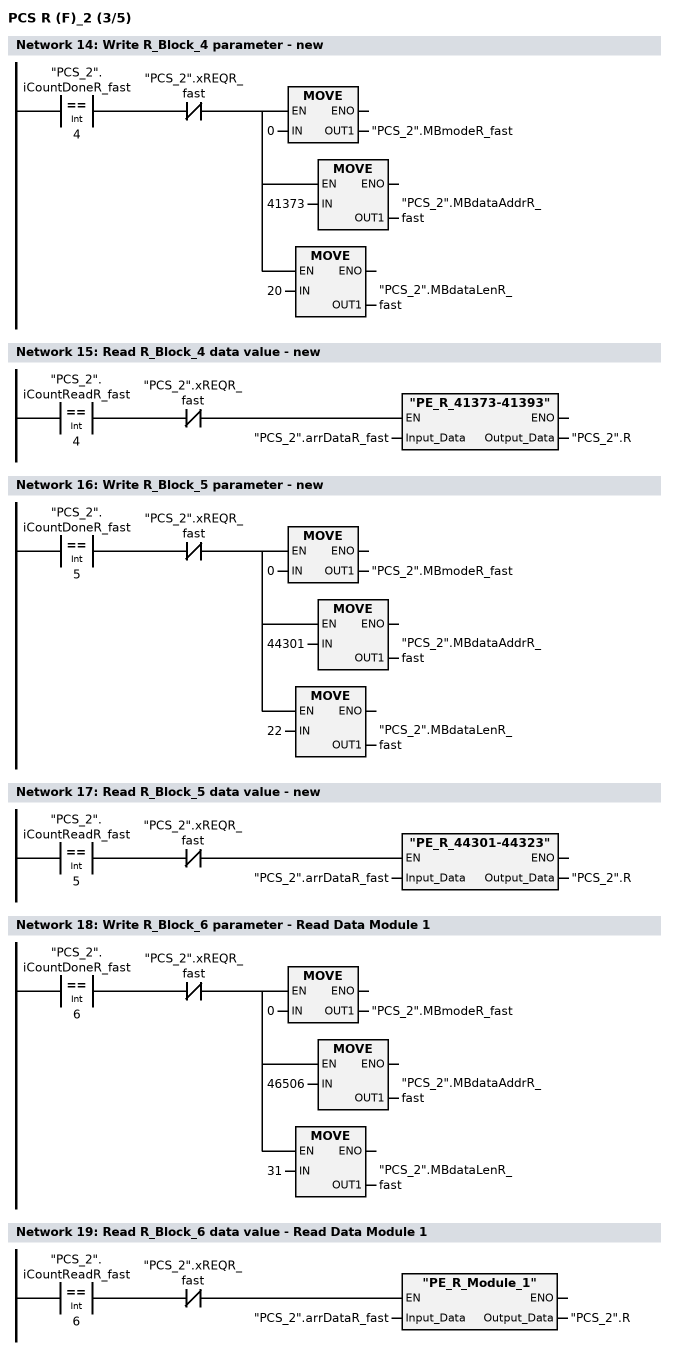
   RUNG wire#powerrail
      { S7_Templates := "SrcType := Int" } EQ_Contact(in1 := "PCS_2".iCountDoneR_fast, in2 := 4)
      I_Contact( "PCS_2".xREQR_fast )
      wire#w1
      Move(in := 0, out1 => "PCS_2".MBmodeR_fast)
   END_RUNG
   RUNG wire#w1
      Move(in := 41373, out1 => "PCS_2".MBdataAddrR_fast)
   END_RUNG
   RUNG wire#w1
      Move(in := 20, out1 => "PCS_2".MBdataLenR_fast)
   END_RUNG
   // the same network as SCL:
   IF ("PCS_2".iCountDoneR_fast = 4) AND NOT "PCS_2".xREQR_fast THEN
       "PCS_2".MBmodeR_fast := 0;
       "PCS_2".MBdataAddrR_fast := 41373;
       "PCS_2".MBdataLenR_fast := 20;
   END_IF;
END_REGION

REGION Network 15: Read R_Block_4 data value - new
   RUNG wire#powerrail
      { S7_Templates := "SrcType := Int" } EQ_Contact(in1 := "PCS_2".iCountReadR_fast, in2 := 4)
      I_Contact( "PCS_2".xREQR_fast )
      "PE_R_41373-41393"(Input_Data := "PCS_2".arrDataR_fast, Output_Data => "PCS_2".R)
   END_RUNG
   // the same network as SCL:
   IF ("PCS_2".iCountReadR_fast = 4) AND NOT "PCS_2".xREQR_fast THEN
       "PE_R_41373-41393"(Input_Data := "PCS_2".arrDataR_fast, Output_Data => "PCS_2".R);
   END_IF;
END_REGION

REGION Network 16: Write R_Block_5 parameter - new
   RUNG wire#powerrail
      { S7_Templates := "SrcType := Int" } EQ_Contact(in1 := "PCS_2".iCountDoneR_fast, in2 := 5)
      I_Contact( "PCS_2".xREQR_fast )
      wire#w1
      Move(in := 0, out1 => "PCS_2".MBmodeR_fast)
   END_RUNG
   RUNG wire#w1
      Move(in := 44301, out1 => "PCS_2".MBdataAddrR_fast)
   END_RUNG
   RUNG wire#w1
      Move(in := 22, out1 => "PCS_2".MBdataLenR_fast)
   END_RUNG
   // the same network as SCL:
   IF ("PCS_2".iCountDoneR_fast = 5) AND NOT "PCS_2".xREQR_fast THEN
       "PCS_2".MBmodeR_fast := 0;
       "PCS_2".MBdataAddrR_fast := 44301;
       "PCS_2".MBdataLenR_fast := 22;
   END_IF;
END_REGION

REGION Network 17: Read R_Block_5 data value - new
   RUNG wire#powerrail
      { S7_Templates := "SrcType := Int" } EQ_Contact(in1 := "PCS_2".iCountReadR_fast, in2 := 5)
      I_Contact( "PCS_2".xREQR_fast )
      "PE_R_44301-44323"(Input_Data := "PCS_2".arrDataR_fast, Output_Data => "PCS_2".R)
   END_RUNG
   // the same network as SCL:
   IF ("PCS_2".iCountReadR_fast = 5) AND NOT "PCS_2".xREQR_fast THEN
       "PE_R_44301-44323"(Input_Data := "PCS_2".arrDataR_fast, Output_Data => "PCS_2".R);
   END_IF;
END_REGION

REGION Network 18: Write R_Block_6 parameter - Read Data Module 1
   RUNG wire#powerrail
      { S7_Templates := "SrcType := Int" } EQ_Contact(in1 := "PCS_2".iCountDoneR_fast, in2 := 6)
      I_Contact( "PCS_2".xREQR_fast )
      wire#w1
      Move(in := 0, out1 => "PCS_2".MBmodeR_fast)
   END_RUNG
   RUNG wire#w1
      Move(in := 46506, out1 => "PCS_2".MBdataAddrR_fast)
   END_RUNG
   RUNG wire#w1
      Move(in := 31, out1 => "PCS_2".MBdataLenR_fast)
   END_RUNG
   // the same network as SCL:
   IF ("PCS_2".iCountDoneR_fast = 6) AND NOT "PCS_2".xREQR_fast THEN
       "PCS_2".MBmodeR_fast := 0;
       "PCS_2".MBdataAddrR_fast := 46506;
       "PCS_2".MBdataLenR_fast := 31;
   END_IF;
END_REGION

REGION Network 19: Read R_Block_6 data value - Read Data Module 1
   RUNG wire#powerrail
      { S7_Templates := "SrcType := Int" } EQ_Contact(in1 := "PCS_2".iCountReadR_fast, in2 := 6)
      I_Contact( "PCS_2".xREQR_fast )
      "PE_R_Module_1"(Input_Data := "PCS_2".arrDataR_fast, Output_Data => "PCS_2".R)
   END_RUNG
   // the same network as SCL:
   IF ("PCS_2".iCountReadR_fast = 6) AND NOT "PCS_2".xREQR_fast THEN
       "PE_R_Module_1"(Input_Data := "PCS_2".arrDataR_fast, Output_Data => "PCS_2".R);
   END_IF;
END_REGION

REGION Network 20: Write R_Block_7 parameter - Read Data Module 2
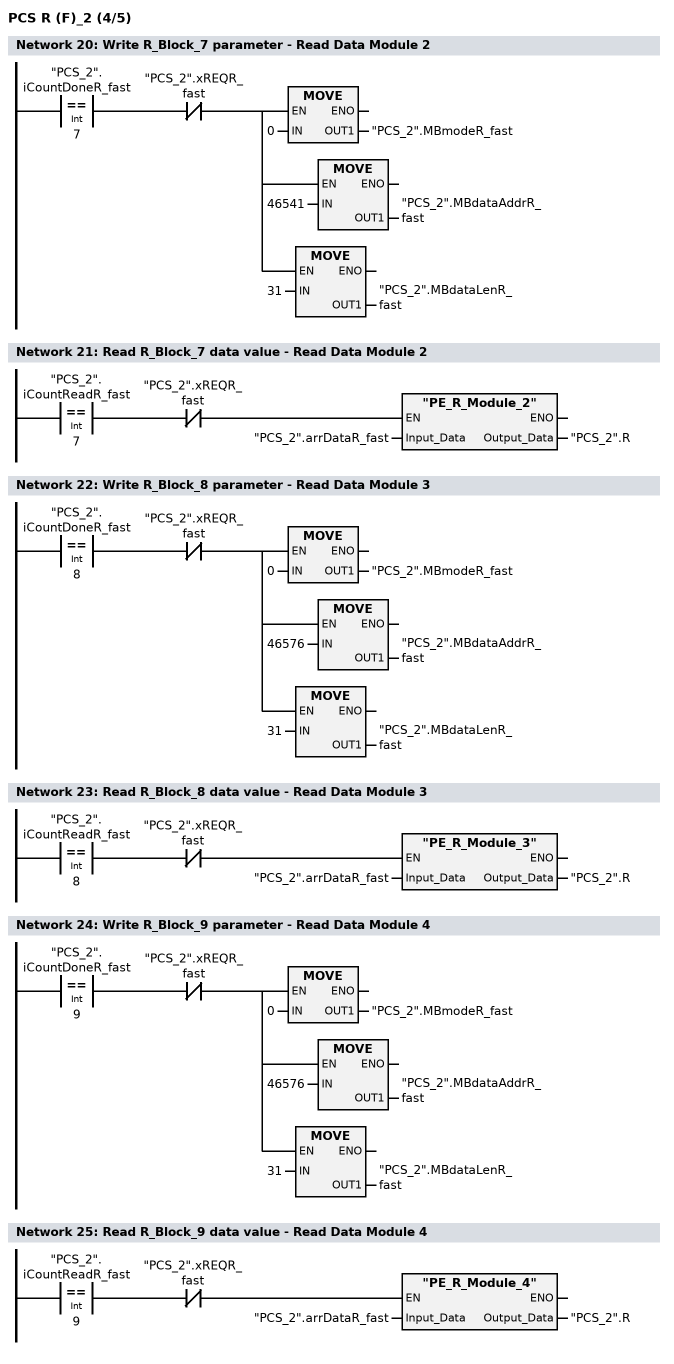
   RUNG wire#powerrail
      { S7_Templates := "SrcType := Int" } EQ_Contact(in1 := "PCS_2".iCountDoneR_fast, in2 := 7)
      I_Contact( "PCS_2".xREQR_fast )
      wire#w1
      Move(in := 0, out1 => "PCS_2".MBmodeR_fast)
   END_RUNG
   RUNG wire#w1
      Move(in := 46541, out1 => "PCS_2".MBdataAddrR_fast)
   END_RUNG
   RUNG wire#w1
      Move(in := 31, out1 => "PCS_2".MBdataLenR_fast)
   END_RUNG
   // the same network as SCL:
   IF ("PCS_2".iCountDoneR_fast = 7) AND NOT "PCS_2".xREQR_fast THEN
       "PCS_2".MBmodeR_fast := 0;
       "PCS_2".MBdataAddrR_fast := 46541;
       "PCS_2".MBdataLenR_fast := 31;
   END_IF;
END_REGION

REGION Network 21: Read R_Block_7 data value - Read Data Module 2
   RUNG wire#powerrail
      { S7_Templates := "SrcType := Int" } EQ_Contact(in1 := "PCS_2".iCountReadR_fast, in2 := 7)
      I_Contact( "PCS_2".xREQR_fast )
      "PE_R_Module_2"(Input_Data := "PCS_2".arrDataR_fast, Output_Data => "PCS_2".R)
   END_RUNG
   // the same network as SCL:
   IF ("PCS_2".iCountReadR_fast = 7) AND NOT "PCS_2".xREQR_fast THEN
       "PE_R_Module_2"(Input_Data := "PCS_2".arrDataR_fast, Output_Data => "PCS_2".R);
   END_IF;
END_REGION

REGION Network 22: Write R_Block_8 parameter - Read Data Module 3
   RUNG wire#powerrail
      { S7_Templates := "SrcType := Int" } EQ_Contact(in1 := "PCS_2".iCountDoneR_fast, in2 := 8)
      I_Contact( "PCS_2".xREQR_fast )
      wire#w1
      Move(in := 0, out1 => "PCS_2".MBmodeR_fast)
   END_RUNG
   RUNG wire#w1
      Move(in := 46576, out1 => "PCS_2".MBdataAddrR_fast)
   END_RUNG
   RUNG wire#w1
      Move(in := 31, out1 => "PCS_2".MBdataLenR_fast)
   END_RUNG
   // the same network as SCL:
   IF ("PCS_2".iCountDoneR_fast = 8) AND NOT "PCS_2".xREQR_fast THEN
       "PCS_2".MBmodeR_fast := 0;
       "PCS_2".MBdataAddrR_fast := 46576;
       "PCS_2".MBdataLenR_fast := 31;
   END_IF;
END_REGION

REGION Network 23: Read R_Block_8 data value - Read Data Module 3
   RUNG wire#powerrail
      { S7_Templates := "SrcType := Int" } EQ_Contact(in1 := "PCS_2".iCountReadR_fast, in2 := 8)
      I_Contact( "PCS_2".xREQR_fast )
      "PE_R_Module_3"(Input_Data := "PCS_2".arrDataR_fast, Output_Data => "PCS_2".R)
   END_RUNG
   // the same network as SCL:
   IF ("PCS_2".iCountReadR_fast = 8) AND NOT "PCS_2".xREQR_fast THEN
       "PE_R_Module_3"(Input_Data := "PCS_2".arrDataR_fast, Output_Data => "PCS_2".R);
   END_IF;
END_REGION

REGION Network 24: Write R_Block_9 parameter - Read Data Module 4
   RUNG wire#powerrail
      { S7_Templates := "SrcType := Int" } EQ_Contact(in1 := "PCS_2".iCountDoneR_fast, in2 := 9)
      I_Contact( "PCS_2".xREQR_fast )
      wire#w1
      Move(in := 0, out1 => "PCS_2".MBmodeR_fast)
   END_RUNG
   RUNG wire#w1
      Move(in := 46576, out1 => "PCS_2".MBdataAddrR_fast)
   END_RUNG
   RUNG wire#w1
      Move(in := 31, out1 => "PCS_2".MBdataLenR_fast)
   END_RUNG
   // the same network as SCL:
   IF ("PCS_2".iCountDoneR_fast = 9) AND NOT "PCS_2".xREQR_fast THEN
       "PCS_2".MBmodeR_fast := 0;
       "PCS_2".MBdataAddrR_fast := 46576;
       "PCS_2".MBdataLenR_fast := 31;
   END_IF;
END_REGION

REGION Network 25: Read R_Block_9 data value - Read Data Module 4
   RUNG wire#powerrail
      { S7_Templates := "SrcType := Int" } EQ_Contact(in1 := "PCS_2".iCountReadR_fast, in2 := 9)
      I_Contact( "PCS_2".xREQR_fast )
      "PE_R_Module_4"(Input_Data := "PCS_2".arrDataR_fast, Output_Data => "PCS_2".R)
   END_RUNG
   // the same network as SCL:
   IF ("PCS_2".iCountReadR_fast = 9) AND NOT "PCS_2".xREQR_fast THEN
       "PE_R_Module_4"(Input_Data := "PCS_2".arrDataR_fast, Output_Data => "PCS_2".R);
   END_IF;
END_REGION

REGION Network 26: Write R_Block_10 parameter - Read Humidity module 1-2-3-4
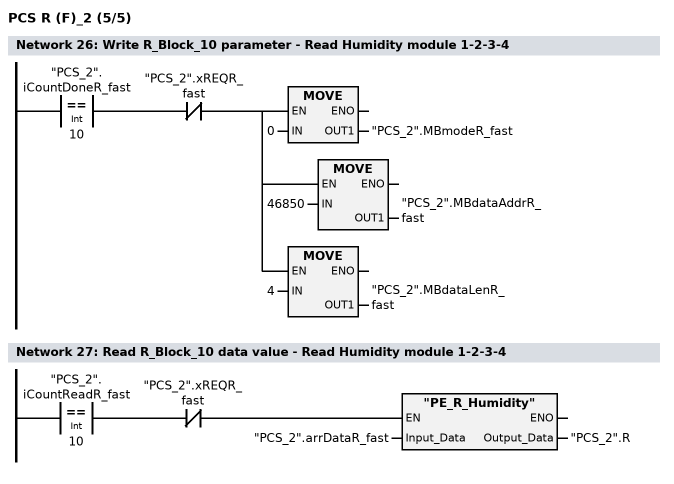
   RUNG wire#powerrail
      { S7_Templates := "SrcType := Int" } EQ_Contact(in1 := "PCS_2".iCountDoneR_fast, in2 := 10)
      I_Contact( "PCS_2".xREQR_fast )
      wire#w1
      Move(in := 0, out1 => "PCS_2".MBmodeR_fast)
   END_RUNG
   RUNG wire#w1
      Move(in := 46850, out1 => "PCS_2".MBdataAddrR_fast)
   END_RUNG
   RUNG wire#w1
      Move(in := 4, out1 => "PCS_2".MBdataLenR_fast)
   END_RUNG
   // the same network as SCL:
   IF ("PCS_2".iCountDoneR_fast = 10) AND NOT "PCS_2".xREQR_fast THEN
       "PCS_2".MBmodeR_fast := 0;
       "PCS_2".MBdataAddrR_fast := 46850;
       "PCS_2".MBdataLenR_fast := 4;
   END_IF;
END_REGION

REGION Network 27: Read R_Block_10 data value - Read Humidity module 1-2-3-4
   RUNG wire#powerrail
      { S7_Templates := "SrcType := Int" } EQ_Contact(in1 := "PCS_2".iCountReadR_fast, in2 := 10)
      I_Contact( "PCS_2".xREQR_fast )
      "PE_R_Humidity"(Input_Data := "PCS_2".arrDataR_fast, Output_Data => "PCS_2".R)
   END_RUNG
   // the same network as SCL:
   IF ("PCS_2".iCountReadR_fast = 10) AND NOT "PCS_2".xREQR_fast THEN
       "PE_R_Humidity"(Input_Data := "PCS_2".arrDataR_fast, Output_Data => "PCS_2".R);
   END_IF;
END_REGION
END_FUNCTION

FUNCTION "PCS R (S)_2" : Void   // FC49, LAD
TITLE = ModBus TCP for PCS Power Electronics
{ S7_Optimized_Access := 'TRUE' }
VERSION : 0.1
// stored: AutoNumber true, IsIECCheckEnabled false, SetENOAutomatically false, UDAEnableTagReadback false
   VAR_TEMP
      rVac : Real;
   END_VAR
   VAR_TEMP   // added for the SCL form of the ladder/FBD networks
      _w1 : Bool;
   END_VAR
BEGIN

REGION Network 1: Function Modbus Client
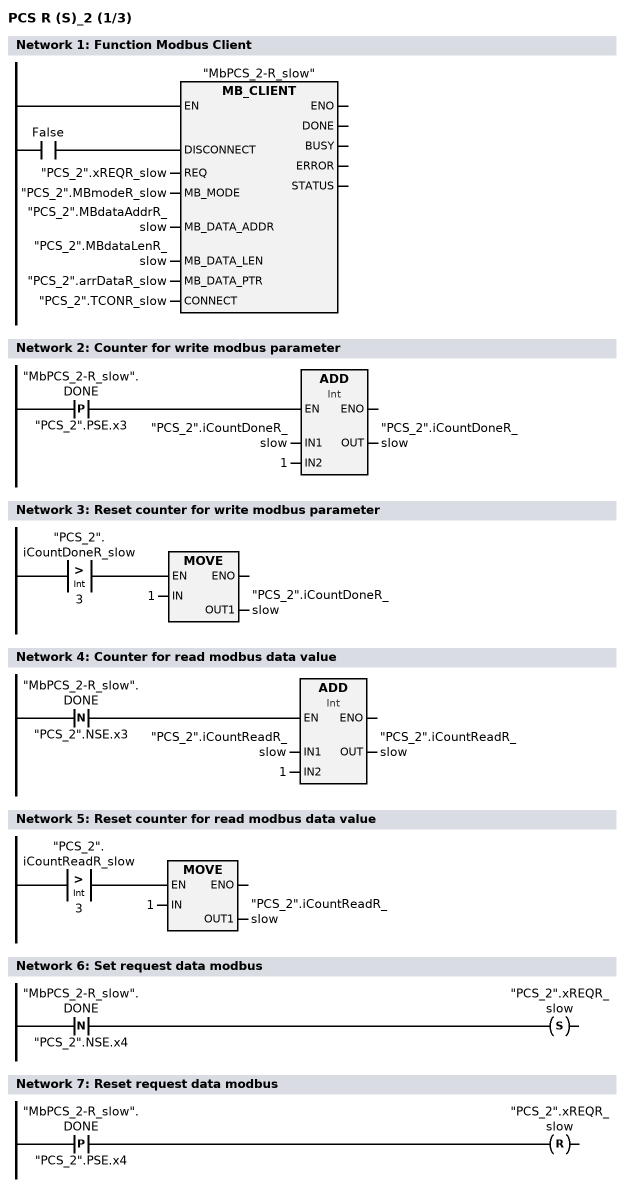
   RUNG wire#powerrail
      "MbPCS_2-R_slow".MB_CLIENT(DISCONNECT := wire#w1, REQ := "PCS_2".xREQR_slow, MB_MODE := "PCS_2".MBmodeR_slow, MB_DATA_ADDR := "PCS_2".MBdataAddrR_slow, MB_DATA_LEN := "PCS_2".MBdataLenR_slow, MB_DATA_PTR := "PCS_2".arrDataR_slow, CONNECT := "PCS_2".TCONR_slow, DONE =>, BUSY =>, ERROR =>, STATUS =>)
   END_RUNG
   RUNG wire#powerrail
      Contact( False )
   END_RUNG wire#w1
   // the same network as SCL:
   "MbPCS_2-R_slow"(DISCONNECT := False,   // MB_CLIENT
                    REQ := "PCS_2".xREQR_slow,
                    MB_MODE := "PCS_2".MBmodeR_slow,
                    MB_DATA_ADDR := "PCS_2".MBdataAddrR_slow,
                    MB_DATA_LEN := "PCS_2".MBdataLenR_slow,
                    MB_DATA_PTR := "PCS_2".arrDataR_slow,
                    CONNECT := "PCS_2".TCONR_slow);
END_REGION

REGION Network 2: Counter for write modbus parameter
   RUNG wire#powerrail
      P_Contact(operand := "MbPCS_2-R_slow".DONE, bit := "PCS_2".PSE.x3)
      { S7_Templates := "SrcType := Int" } Add(in1 := "PCS_2".iCountDoneR_slow, in2 := 1, out => "PCS_2".iCountDoneR_slow)
   END_RUNG
   // the same network as SCL:
   #_w1 := "MbPCS_2-R_slow".DONE AND NOT "PCS_2".PSE.x3;   // rising edge of "MbPCS_2-R_slow".DONE
   "PCS_2".PSE.x3 := "MbPCS_2-R_slow".DONE;
   IF #_w1 THEN "PCS_2".iCountDoneR_slow := "PCS_2".iCountDoneR_slow + 1; END_IF;
END_REGION

REGION Network 3: Reset counter for write modbus parameter
   RUNG wire#powerrail
      { S7_Templates := "SrcType := Int" } GT_Contact(in1 := "PCS_2".iCountDoneR_slow, in2 := 3)
      Move(in := 1, out1 => "PCS_2".iCountDoneR_slow)
   END_RUNG
   // the same network as SCL:
   IF "PCS_2".iCountDoneR_slow > 3 THEN "PCS_2".iCountDoneR_slow := 1; END_IF;
END_REGION

REGION Network 4: Counter for read modbus data value
   RUNG wire#powerrail
      N_Contact(operand := "MbPCS_2-R_slow".DONE, bit := "PCS_2".NSE.x3)
      { S7_Templates := "SrcType := Int" } Add(in1 := "PCS_2".iCountReadR_slow, in2 := 1, out => "PCS_2".iCountReadR_slow)
   END_RUNG
   // the same network as SCL:
   #_w1 := NOT "MbPCS_2-R_slow".DONE AND "PCS_2".NSE.x3;   // falling edge of "MbPCS_2-R_slow".DONE
   "PCS_2".NSE.x3 := "MbPCS_2-R_slow".DONE;
   IF #_w1 THEN "PCS_2".iCountReadR_slow := "PCS_2".iCountReadR_slow + 1; END_IF;
END_REGION

REGION Network 5: Reset counter for read modbus data value
   RUNG wire#powerrail
      { S7_Templates := "SrcType := Int" } GT_Contact(in1 := "PCS_2".iCountReadR_slow, in2 := 3)
      Move(in := 1, out1 => "PCS_2".iCountReadR_slow)
   END_RUNG
   // the same network as SCL:
   IF "PCS_2".iCountReadR_slow > 3 THEN "PCS_2".iCountReadR_slow := 1; END_IF;
END_REGION

REGION Network 6: Set request data modbus
   RUNG wire#powerrail
      N_Contact(operand := "MbPCS_2-R_slow".DONE, bit := "PCS_2".NSE.x4)
      S_Coil( "PCS_2".xREQR_slow )
   END_RUNG
   // the same network as SCL:
   #_w1 := NOT "MbPCS_2-R_slow".DONE AND "PCS_2".NSE.x4;   // falling edge of "MbPCS_2-R_slow".DONE
   "PCS_2".NSE.x4 := "MbPCS_2-R_slow".DONE;
   IF #_w1 THEN "PCS_2".xREQR_slow := TRUE; END_IF;
END_REGION

REGION Network 7: Reset request data modbus
   RUNG wire#powerrail
      P_Contact(operand := "MbPCS_2-R_slow".DONE, bit := "PCS_2".PSE.x4)
      R_Coil( "PCS_2".xREQR_slow )
   END_RUNG
   // the same network as SCL:
   #_w1 := "MbPCS_2-R_slow".DONE AND NOT "PCS_2".PSE.x4;   // rising edge of "MbPCS_2-R_slow".DONE
   "PCS_2".PSE.x4 := "MbPCS_2-R_slow".DONE;
   IF #_w1 THEN "PCS_2".xREQR_slow := FALSE; END_IF;
END_REGION

REGION Network 9: Write RW_Block1 parameter - da controllare password
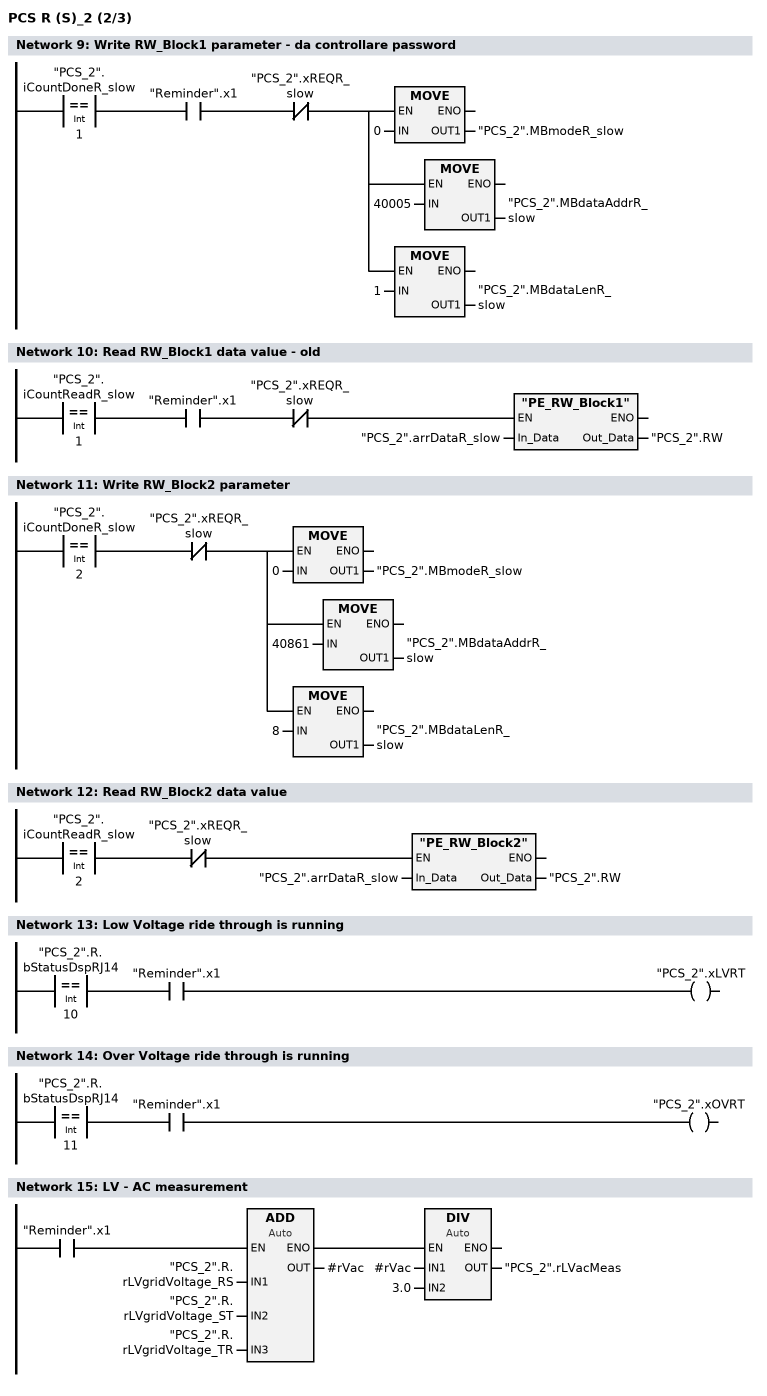
   RUNG wire#powerrail
      { S7_Templates := "SrcType := Int" } EQ_Contact(in1 := "PCS_2".iCountDoneR_slow, in2 := 1)
      Contact( "Reminder".x1 )
      I_Contact( "PCS_2".xREQR_slow )
      wire#w1
      Move(in := 0, out1 => "PCS_2".MBmodeR_slow)
   END_RUNG
   RUNG wire#w1
      Move(in := 40005, out1 => "PCS_2".MBdataAddrR_slow)
   END_RUNG
   RUNG wire#w1
      Move(in := 1, out1 => "PCS_2".MBdataLenR_slow)
   END_RUNG
   // the same network as SCL:
   IF ("PCS_2".iCountDoneR_slow = 1) AND "Reminder".x1 AND NOT "PCS_2".xREQR_slow THEN
       "PCS_2".MBmodeR_slow := 0;
       "PCS_2".MBdataAddrR_slow := 40005;
       "PCS_2".MBdataLenR_slow := 1;
   END_IF;
END_REGION

REGION Network 10: Read RW_Block1 data value - old
   RUNG wire#powerrail
      { S7_Templates := "SrcType := Int" } EQ_Contact(in1 := "PCS_2".iCountReadR_slow, in2 := 1)
      Contact( "Reminder".x1 )
      I_Contact( "PCS_2".xREQR_slow )
      "PE_RW_Block1"(In_Data := "PCS_2".arrDataR_slow, Out_Data => "PCS_2".RW)
   END_RUNG
   // the same network as SCL:
   IF ("PCS_2".iCountReadR_slow = 1) AND "Reminder".x1 AND NOT "PCS_2".xREQR_slow THEN
       "PE_RW_Block1"(In_Data := "PCS_2".arrDataR_slow, Out_Data => "PCS_2".RW);
   END_IF;
END_REGION

REGION Network 11: Write RW_Block2 parameter
   RUNG wire#powerrail
      { S7_Templates := "SrcType := Int" } EQ_Contact(in1 := "PCS_2".iCountDoneR_slow, in2 := 2)
      I_Contact( "PCS_2".xREQR_slow )
      wire#w1
      Move(in := 0, out1 => "PCS_2".MBmodeR_slow)
   END_RUNG
   RUNG wire#w1
      Move(in := 40861, out1 => "PCS_2".MBdataAddrR_slow)
   END_RUNG
   RUNG wire#w1
      Move(in := 8, out1 => "PCS_2".MBdataLenR_slow)
   END_RUNG
   // the same network as SCL:
   IF ("PCS_2".iCountDoneR_slow = 2) AND NOT "PCS_2".xREQR_slow THEN
       "PCS_2".MBmodeR_slow := 0;
       "PCS_2".MBdataAddrR_slow := 40861;
       "PCS_2".MBdataLenR_slow := 8;
   END_IF;
END_REGION

REGION Network 12: Read RW_Block2 data value
   RUNG wire#powerrail
      { S7_Templates := "SrcType := Int" } EQ_Contact(in1 := "PCS_2".iCountReadR_slow, in2 := 2)
      I_Contact( "PCS_2".xREQR_slow )
      "PE_RW_Block2"(In_Data := "PCS_2".arrDataR_slow, Out_Data => "PCS_2".RW)
   END_RUNG
   // the same network as SCL:
   IF ("PCS_2".iCountReadR_slow = 2) AND NOT "PCS_2".xREQR_slow THEN
       "PE_RW_Block2"(In_Data := "PCS_2".arrDataR_slow, Out_Data => "PCS_2".RW);
   END_IF;
END_REGION

REGION Network 13: Low Voltage ride through is running
   RUNG wire#powerrail
      { S7_Templates := "SrcType := Int" } EQ_Contact(in1 := "PCS_2".R.bStatusDspRJ14, in2 := 10)
      Contact( "Reminder".x1 )
      Coil( "PCS_2".xLVRT )
   END_RUNG
   // the same network as SCL:
   "PCS_2".xLVRT := ("PCS_2".R.bStatusDspRJ14 = 10) AND "Reminder".x1;
END_REGION

REGION Network 14: Over Voltage ride through is running
   RUNG wire#powerrail
      { S7_Templates := "SrcType := Int" } EQ_Contact(in1 := "PCS_2".R.bStatusDspRJ14, in2 := 11)
      Contact( "Reminder".x1 )
      Coil( "PCS_2".xOVRT )
   END_RUNG
   // the same network as SCL:
   "PCS_2".xOVRT := ("PCS_2".R.bStatusDspRJ14 = 11) AND "Reminder".x1;
END_REGION

REGION Network 15: LV - AC measurement
   RUNG wire#powerrail
      Contact( "Reminder".x1 )
      Add(in1 := "PCS_2".R.rLVgridVoltage_RS, in2 := "PCS_2".R.rLVgridVoltage_ST, in3 := "PCS_2".R.rLVgridVoltage_TR, out => #rVac)
      Div(in1 := #rVac, in2 := 3.0, out => "PCS_2".rLVacMeas)
   END_RUNG
   // the same network as SCL:
   IF "Reminder".x1 THEN
       #rVac := "PCS_2".R.rLVgridVoltage_RS + "PCS_2".R.rLVgridVoltage_ST + "PCS_2".R.rLVgridVoltage_TR;
       "PCS_2".rLVacMeas := #rVac / 3.0;
   END_IF;
END_REGION

REGION Network 16: MV - AC measurement
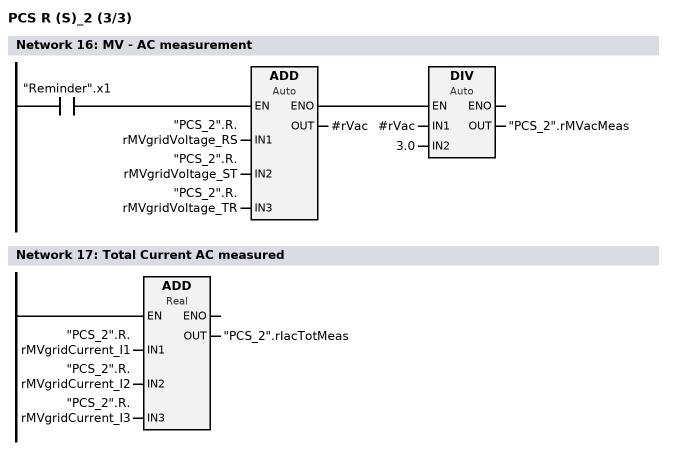
   RUNG wire#powerrail
      Contact( "Reminder".x1 )
      Add(in1 := "PCS_2".R.rMVgridVoltage_RS, in2 := "PCS_2".R.rMVgridVoltage_ST, in3 := "PCS_2".R.rMVgridVoltage_TR, out => #rVac)
      Div(in1 := #rVac, in2 := 3.0, out => "PCS_2".rMVacMeas)
   END_RUNG
   // the same network as SCL:
   IF "Reminder".x1 THEN
       #rVac := "PCS_2".R.rMVgridVoltage_RS + "PCS_2".R.rMVgridVoltage_ST + "PCS_2".R.rMVgridVoltage_TR;
       "PCS_2".rMVacMeas := #rVac / 3.0;
   END_IF;
END_REGION

REGION Network 17: Total Current AC measured
   RUNG wire#powerrail
      { S7_Templates := "SrcType := Real" } Add(in1 := "PCS_2".R.rMVgridCurrent_I1, in2 := "PCS_2".R.rMVgridCurrent_I2, in3 := "PCS_2".R.rMVgridCurrent_I3, out => "PCS_2".rIacTotMeas)
   END_RUNG
   // the same network as SCL:
   "PCS_2".rIacTotMeas := "PCS_2".R.rMVgridCurrent_I1 + "PCS_2".R.rMVgridCurrent_I2 + "PCS_2".R.rMVgridCurrent_I3;
END_REGION
END_FUNCTION

FUNCTION "PCS W (F)_2" : Void   // FC42, LAD
TITLE = ModBus TCP for PCS Power Electronics
{ S7_Optimized_Access := 'TRUE' }
VERSION : 0.1
// stored: AutoNumber false, IsIECCheckEnabled false, SetENOAutomatically false, UDAEnableTagReadback false
   VAR_TEMP
      rSS1PacRef : Real;
      rSS2PacRef : Real;
      rSS1QacRef : Real;
      rSS2QacRef : Real;
      rSnHalfPE : Real;
      rQacRef : Real;
      uiQacRef : UInt;
   END_VAR
   VAR_TEMP   // added for the SCL form of the ladder/FBD networks
      _w1 : Bool;
   END_VAR
BEGIN

REGION Network 1: Function Modbus Client
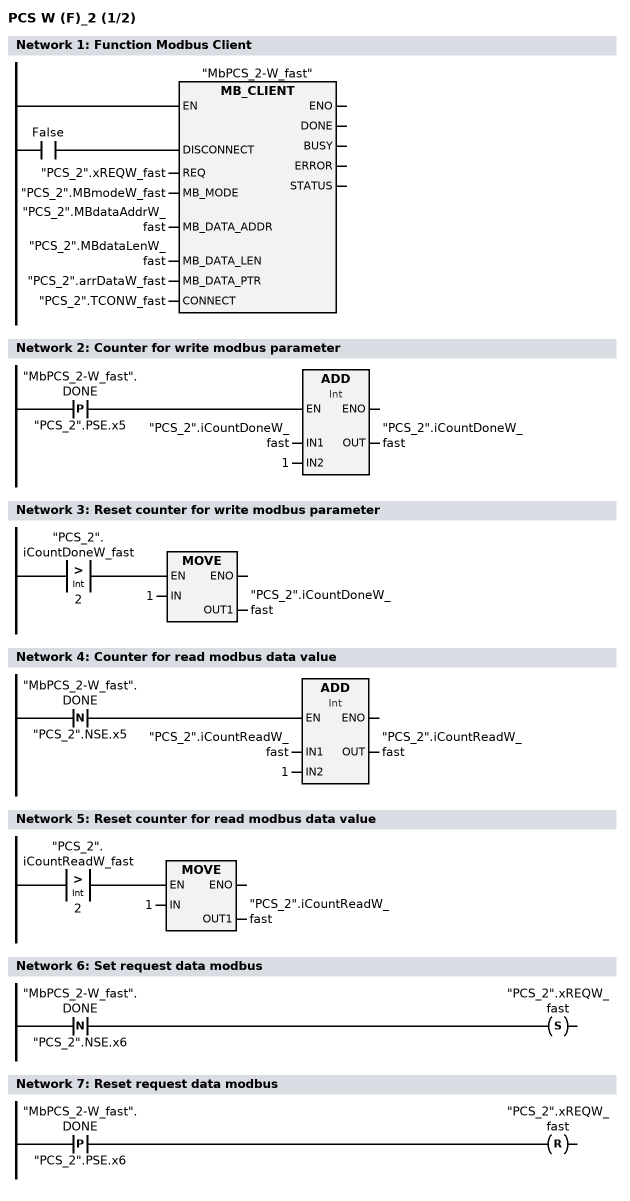
   RUNG wire#powerrail
      "MbPCS_2-W_fast".MB_CLIENT(DISCONNECT := wire#w1, REQ := "PCS_2".xREQW_fast, MB_MODE := "PCS_2".MBmodeW_fast, MB_DATA_ADDR := "PCS_2".MBdataAddrW_fast, MB_DATA_LEN := "PCS_2".MBdataLenW_fast, MB_DATA_PTR := "PCS_2".arrDataW_fast, CONNECT := "PCS_2".TCONW_fast, DONE =>, BUSY =>, ERROR =>, STATUS =>)
   END_RUNG
   RUNG wire#powerrail
      Contact( False )
   END_RUNG wire#w1
   // the same network as SCL:
   "MbPCS_2-W_fast"(DISCONNECT := False,   // MB_CLIENT
                    REQ := "PCS_2".xREQW_fast,
                    MB_MODE := "PCS_2".MBmodeW_fast,
                    MB_DATA_ADDR := "PCS_2".MBdataAddrW_fast,
                    MB_DATA_LEN := "PCS_2".MBdataLenW_fast,
                    MB_DATA_PTR := "PCS_2".arrDataW_fast,
                    CONNECT := "PCS_2".TCONW_fast);
END_REGION

REGION Network 2: Counter for write modbus parameter
   RUNG wire#powerrail
      P_Contact(operand := "MbPCS_2-W_fast".DONE, bit := "PCS_2".PSE.x5)
      { S7_Templates := "SrcType := Int" } Add(in1 := "PCS_2".iCountDoneW_fast, in2 := 1, out => "PCS_2".iCountDoneW_fast)
   END_RUNG
   // the same network as SCL:
   #_w1 := "MbPCS_2-W_fast".DONE AND NOT "PCS_2".PSE.x5;   // rising edge of "MbPCS_2-W_fast".DONE
   "PCS_2".PSE.x5 := "MbPCS_2-W_fast".DONE;
   IF #_w1 THEN "PCS_2".iCountDoneW_fast := "PCS_2".iCountDoneW_fast + 1; END_IF;
END_REGION

REGION Network 3: Reset counter for write modbus parameter
   RUNG wire#powerrail
      { S7_Templates := "SrcType := Int" } GT_Contact(in1 := "PCS_2".iCountDoneW_fast, in2 := 2)
      Move(in := 1, out1 => "PCS_2".iCountDoneW_fast)
   END_RUNG
   // the same network as SCL:
   IF "PCS_2".iCountDoneW_fast > 2 THEN "PCS_2".iCountDoneW_fast := 1; END_IF;
END_REGION

REGION Network 4: Counter for read modbus data value
   RUNG wire#powerrail
      N_Contact(operand := "MbPCS_2-W_fast".DONE, bit := "PCS_2".NSE.x5)
      { S7_Templates := "SrcType := Int" } Add(in1 := "PCS_2".iCountReadW_fast, in2 := 1, out => "PCS_2".iCountReadW_fast)
   END_RUNG
   // the same network as SCL:
   #_w1 := NOT "MbPCS_2-W_fast".DONE AND "PCS_2".NSE.x5;   // falling edge of "MbPCS_2-W_fast".DONE
   "PCS_2".NSE.x5 := "MbPCS_2-W_fast".DONE;
   IF #_w1 THEN "PCS_2".iCountReadW_fast := "PCS_2".iCountReadW_fast + 1; END_IF;
END_REGION

REGION Network 5: Reset counter for read modbus data value
   RUNG wire#powerrail
      { S7_Templates := "SrcType := Int" } GT_Contact(in1 := "PCS_2".iCountReadW_fast, in2 := 2)
      Move(in := 1, out1 => "PCS_2".iCountReadW_fast)
   END_RUNG
   // the same network as SCL:
   IF "PCS_2".iCountReadW_fast > 2 THEN "PCS_2".iCountReadW_fast := 1; END_IF;
END_REGION

REGION Network 6: Set request data modbus
   RUNG wire#powerrail
      N_Contact(operand := "MbPCS_2-W_fast".DONE, bit := "PCS_2".NSE.x6)
      S_Coil( "PCS_2".xREQW_fast )
   END_RUNG
   // the same network as SCL:
   #_w1 := NOT "MbPCS_2-W_fast".DONE AND "PCS_2".NSE.x6;   // falling edge of "MbPCS_2-W_fast".DONE
   "PCS_2".NSE.x6 := "MbPCS_2-W_fast".DONE;
   IF #_w1 THEN "PCS_2".xREQW_fast := TRUE; END_IF;
END_REGION

REGION Network 7: Reset request data modbus
   RUNG wire#powerrail
      P_Contact(operand := "MbPCS_2-W_fast".DONE, bit := "PCS_2".PSE.x6)
      R_Coil( "PCS_2".xREQW_fast )
   END_RUNG
   // the same network as SCL:
   #_w1 := "MbPCS_2-W_fast".DONE AND NOT "PCS_2".PSE.x6;   // rising edge of "MbPCS_2-W_fast".DONE
   "PCS_2".PSE.x6 := "MbPCS_2-W_fast".DONE;
   IF #_w1 THEN "PCS_2".xREQW_fast := FALSE; END_IF;
END_REGION

REGION Network 9: Write Active Power Reference
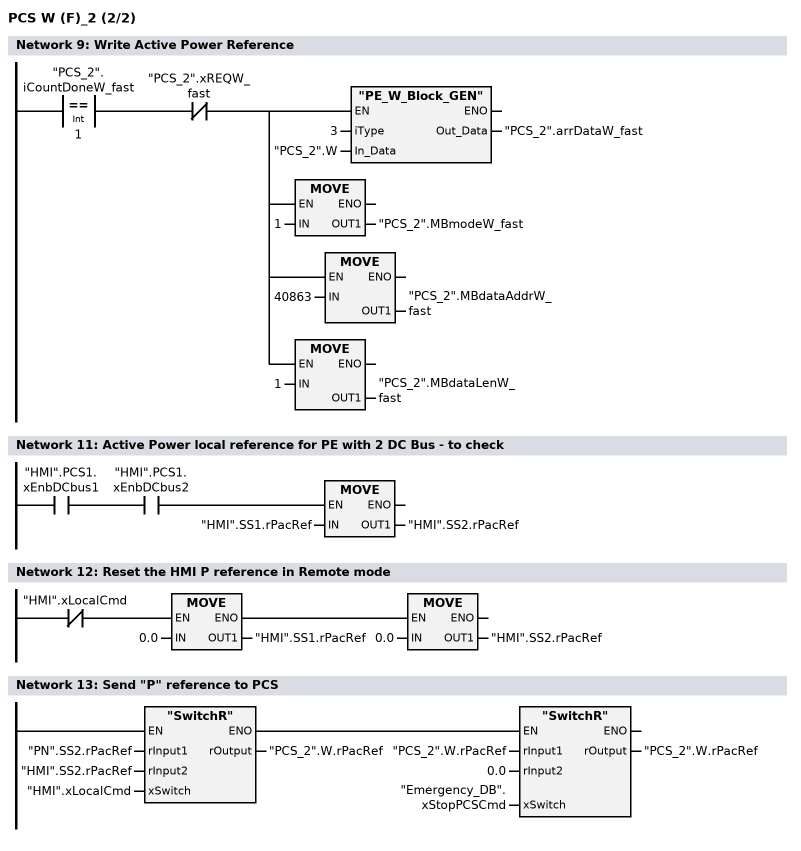
   RUNG wire#powerrail
      { S7_Templates := "SrcType := Int" } EQ_Contact(in1 := "PCS_2".iCountDoneW_fast, in2 := 1)
      I_Contact( "PCS_2".xREQW_fast )
      wire#w1
      "PE_W_Block_GEN"(iType := 3, In_Data := "PCS_2".W, Out_Data => "PCS_2".arrDataW_fast)
   END_RUNG
   RUNG wire#w1
      Move(in := 1, out1 => "PCS_2".MBmodeW_fast)
   END_RUNG
   RUNG wire#w1
      Move(in := 40863, out1 => "PCS_2".MBdataAddrW_fast)
   END_RUNG
   RUNG wire#w1
      Move(in := 1, out1 => "PCS_2".MBdataLenW_fast)
   END_RUNG
   // the same network as SCL:
   #_w1 := ("PCS_2".iCountDoneW_fast = 1) AND NOT "PCS_2".xREQW_fast;
   IF #_w1 THEN
       "PE_W_Block_GEN"(iType := 3, In_Data := "PCS_2".W, Out_Data => "PCS_2".arrDataW_fast);
       "PCS_2".MBmodeW_fast := 1;
       "PCS_2".MBdataAddrW_fast := 40863;
       "PCS_2".MBdataLenW_fast := 1;
   END_IF;
END_REGION

REGION Network 11: Active Power local reference for PE with 2 DC Bus - to check
   RUNG wire#powerrail
      Contact( "HMI".PCS1.xEnbDCbus1 )
      Contact( "HMI".PCS1.xEnbDCbus2 )
      Move(in := "HMI".SS1.rPacRef, out1 => "HMI".SS2.rPacRef)
   END_RUNG
   // the same network as SCL:
   IF "HMI".PCS1.xEnbDCbus1 AND "HMI".PCS1.xEnbDCbus2 THEN "HMI".SS2.rPacRef := "HMI".SS1.rPacRef; END_IF;
END_REGION

REGION Network 12: Reset the HMI P reference in Remote mode
   RUNG wire#powerrail
      I_Contact( "HMI".xLocalCmd )
      Move(in := 0.0, out1 => "HMI".SS1.rPacRef)
      Move(in := 0.0, out1 => "HMI".SS2.rPacRef)
   END_RUNG
   // the same network as SCL:
   IF NOT "HMI".xLocalCmd THEN
       "HMI".SS1.rPacRef := 0.0;
       "HMI".SS2.rPacRef := 0.0;
   END_IF;
END_REGION

REGION Network 13: Send "P" reference to PCS
   RUNG wire#powerrail
      "SwitchR"(rInput1 := "PN".SS2.rPacRef, rInput2 := "HMI".SS2.rPacRef, xSwitch := "HMI".xLocalCmd, rOutput => "PCS_2".W.rPacRef)
      "SwitchR"(rInput1 := "PCS_2".W.rPacRef, rInput2 := 0.0, xSwitch := "Emergency_DB".xStopPCSCmd, rOutput => "PCS_2".W.rPacRef)
   END_RUNG
   // the same network as SCL:
   "SwitchR"(rInput1 := "PN".SS2.rPacRef,
             rInput2 := "HMI".SS2.rPacRef,
             xSwitch := "HMI".xLocalCmd,
             rOutput => "PCS_2".W.rPacRef,
             ENO => #_w1);
   IF #_w1 THEN
       "SwitchR"(rInput1 := "PCS_2".W.rPacRef,
                 rInput2 := 0.0,
                 xSwitch := "Emergency_DB".xStopPCSCmd,
                 rOutput => "PCS_2".W.rPacRef);
   END_IF;
END_REGION
END_FUNCTION

FUNCTION "PCS W (S)_2" : Void   // FC52, LAD
TITLE = ModBus TCP for PCS Power Electronics
{ S7_Optimized_Access := 'TRUE' }
VERSION : 0.1
// stored: AutoNumber true, IsIECCheckEnabled false, SetENOAutomatically false, UDAEnableTagReadback false
   VAR_TEMP
      rSS1PacRef : Real;
      rSS2PacRef : Real;
      rSS1QacRef : Real;
      rSS2QacRef : Real;
      rSnHalfPE : Real;
      rQacRef : Real;
      uiQacRef : UInt;
   END_VAR
   VAR_TEMP   // added for the SCL form of the ladder/FBD networks
      _w1 : Bool;
   END_VAR
BEGIN

REGION Network 1: Function Modbus Client
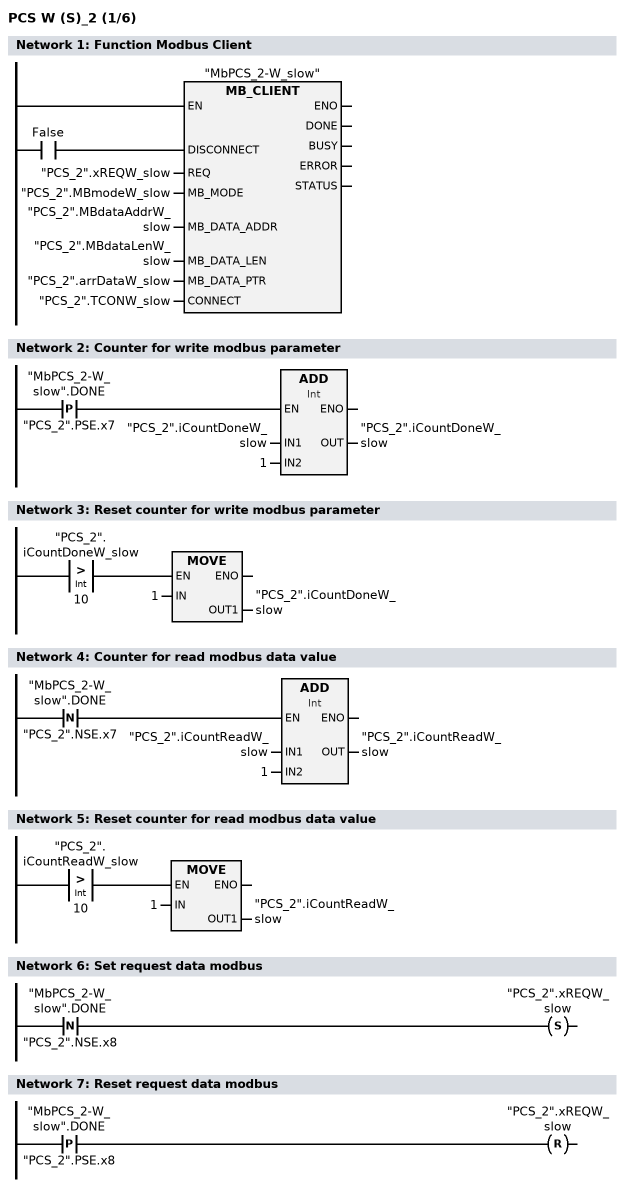
   RUNG wire#powerrail
      "MbPCS_2-W_slow".MB_CLIENT(DISCONNECT := wire#w1, REQ := "PCS_2".xREQW_slow, MB_MODE := "PCS_2".MBmodeW_slow, MB_DATA_ADDR := "PCS_2".MBdataAddrW_slow, MB_DATA_LEN := "PCS_2".MBdataLenW_slow, MB_DATA_PTR := "PCS_2".arrDataW_slow, CONNECT := "PCS_2".TCONW_slow, DONE =>, BUSY =>, ERROR =>, STATUS =>)
   END_RUNG
   RUNG wire#powerrail
      Contact( False )
   END_RUNG wire#w1
   // the same network as SCL:
   "MbPCS_2-W_slow"(DISCONNECT := False,   // MB_CLIENT
                    REQ := "PCS_2".xREQW_slow,
                    MB_MODE := "PCS_2".MBmodeW_slow,
                    MB_DATA_ADDR := "PCS_2".MBdataAddrW_slow,
                    MB_DATA_LEN := "PCS_2".MBdataLenW_slow,
                    MB_DATA_PTR := "PCS_2".arrDataW_slow,
                    CONNECT := "PCS_2".TCONW_slow);
END_REGION

REGION Network 2: Counter for write modbus parameter
   RUNG wire#powerrail
      P_Contact(operand := "MbPCS_2-W_slow".DONE, bit := "PCS_2".PSE.x7)
      { S7_Templates := "SrcType := Int" } Add(in1 := "PCS_2".iCountDoneW_slow, in2 := 1, out => "PCS_2".iCountDoneW_slow)
   END_RUNG
   // the same network as SCL:
   #_w1 := "MbPCS_2-W_slow".DONE AND NOT "PCS_2".PSE.x7;   // rising edge of "MbPCS_2-W_slow".DONE
   "PCS_2".PSE.x7 := "MbPCS_2-W_slow".DONE;
   IF #_w1 THEN "PCS_2".iCountDoneW_slow := "PCS_2".iCountDoneW_slow + 1; END_IF;
END_REGION

REGION Network 3: Reset counter for write modbus parameter
   RUNG wire#powerrail
      { S7_Templates := "SrcType := Int" } GT_Contact(in1 := "PCS_2".iCountDoneW_slow, in2 := 10)
      Move(in := 1, out1 => "PCS_2".iCountDoneW_slow)
   END_RUNG
   // the same network as SCL:
   IF "PCS_2".iCountDoneW_slow > 10 THEN "PCS_2".iCountDoneW_slow := 1; END_IF;
END_REGION

REGION Network 4: Counter for read modbus data value
   RUNG wire#powerrail
      N_Contact(operand := "MbPCS_2-W_slow".DONE, bit := "PCS_2".NSE.x7)
      { S7_Templates := "SrcType := Int" } Add(in1 := "PCS_2".iCountReadW_slow, in2 := 1, out => "PCS_2".iCountReadW_slow)
   END_RUNG
   // the same network as SCL:
   #_w1 := NOT "MbPCS_2-W_slow".DONE AND "PCS_2".NSE.x7;   // falling edge of "MbPCS_2-W_slow".DONE
   "PCS_2".NSE.x7 := "MbPCS_2-W_slow".DONE;
   IF #_w1 THEN "PCS_2".iCountReadW_slow := "PCS_2".iCountReadW_slow + 1; END_IF;
END_REGION

REGION Network 5: Reset counter for read modbus data value
   RUNG wire#powerrail
      { S7_Templates := "SrcType := Int" } GT_Contact(in1 := "PCS_2".iCountReadW_slow, in2 := 10)
      Move(in := 1, out1 => "PCS_2".iCountReadW_slow)
   END_RUNG
   // the same network as SCL:
   IF "PCS_2".iCountReadW_slow > 10 THEN "PCS_2".iCountReadW_slow := 1; END_IF;
END_REGION

REGION Network 6: Set request data modbus
   RUNG wire#powerrail
      N_Contact(operand := "MbPCS_2-W_slow".DONE, bit := "PCS_2".NSE.x8)
      S_Coil( "PCS_2".xREQW_slow )
   END_RUNG
   // the same network as SCL:
   #_w1 := NOT "MbPCS_2-W_slow".DONE AND "PCS_2".NSE.x8;   // falling edge of "MbPCS_2-W_slow".DONE
   "PCS_2".NSE.x8 := "MbPCS_2-W_slow".DONE;
   IF #_w1 THEN "PCS_2".xREQW_slow := TRUE; END_IF;
END_REGION

REGION Network 7: Reset request data modbus
   RUNG wire#powerrail
      P_Contact(operand := "MbPCS_2-W_slow".DONE, bit := "PCS_2".PSE.x8)
      R_Coil( "PCS_2".xREQW_slow )
   END_RUNG
   // the same network as SCL:
   #_w1 := "MbPCS_2-W_slow".DONE AND NOT "PCS_2".PSE.x8;   // rising edge of "MbPCS_2-W_slow".DONE
   "PCS_2".PSE.x8 := "MbPCS_2-W_slow".DONE;
   IF #_w1 THEN "PCS_2".xREQW_slow := FALSE; END_IF;
END_REGION

REGION Network 9: Write W_Block1 parameter - pwd to check
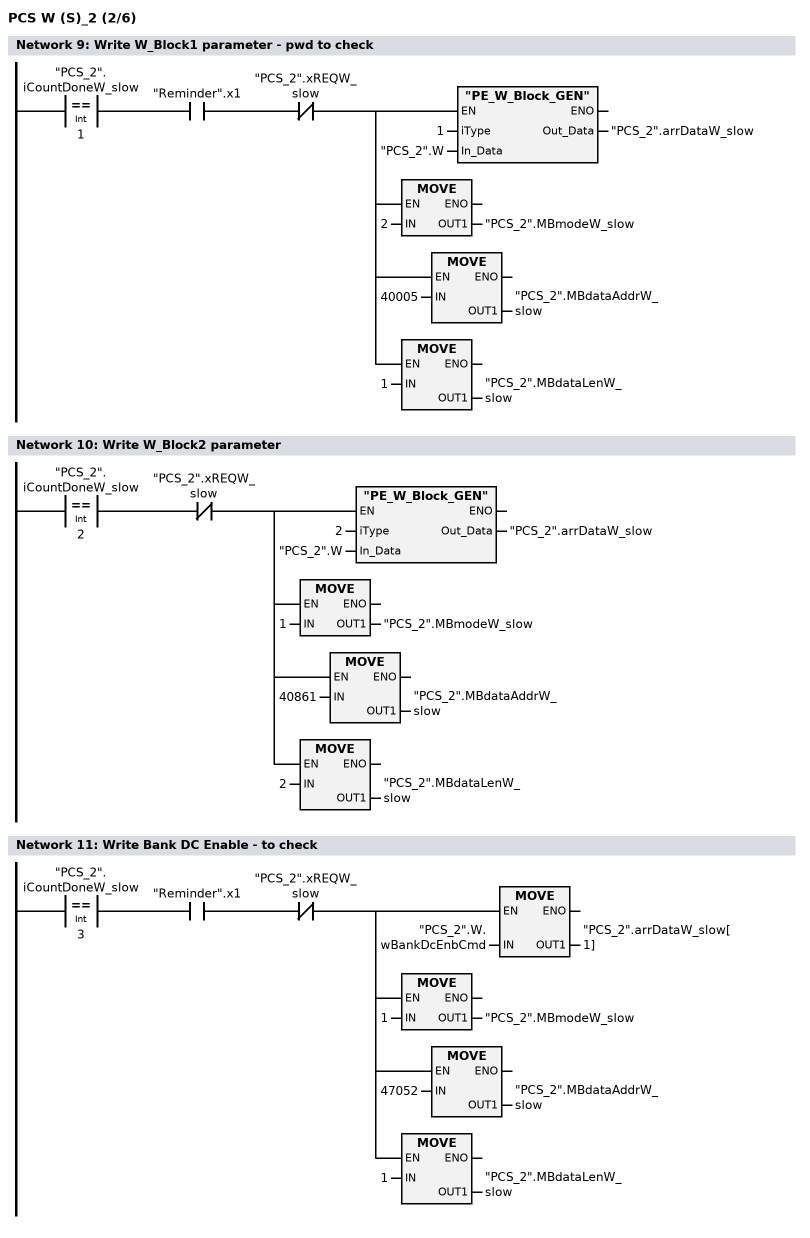
   RUNG wire#powerrail
      { S7_Templates := "SrcType := Int" } EQ_Contact(in1 := "PCS_2".iCountDoneW_slow, in2 := 1)
      Contact( "Reminder".x1 )
      I_Contact( "PCS_2".xREQW_slow )
      wire#w1
      "PE_W_Block_GEN"(iType := 1, In_Data := "PCS_2".W, Out_Data => "PCS_2".arrDataW_slow)
   END_RUNG
   RUNG wire#w1
      Move(in := 2, out1 => "PCS_2".MBmodeW_slow)
   END_RUNG
   RUNG wire#w1
      Move(in := 40005, out1 => "PCS_2".MBdataAddrW_slow)
   END_RUNG
   RUNG wire#w1
      Move(in := 1, out1 => "PCS_2".MBdataLenW_slow)
   END_RUNG
   // the same network as SCL:
   #_w1 := ("PCS_2".iCountDoneW_slow = 1) AND "Reminder".x1 AND NOT "PCS_2".xREQW_slow;
   IF #_w1 THEN
       "PE_W_Block_GEN"(iType := 1, In_Data := "PCS_2".W, Out_Data => "PCS_2".arrDataW_slow);
       "PCS_2".MBmodeW_slow := 2;
       "PCS_2".MBdataAddrW_slow := 40005;
       "PCS_2".MBdataLenW_slow := 1;
   END_IF;
END_REGION

REGION Network 10: Write W_Block2 parameter
   RUNG wire#powerrail
      { S7_Templates := "SrcType := Int" } EQ_Contact(in1 := "PCS_2".iCountDoneW_slow, in2 := 2)
      I_Contact( "PCS_2".xREQW_slow )
      wire#w1
      "PE_W_Block_GEN"(iType := 2, In_Data := "PCS_2".W, Out_Data => "PCS_2".arrDataW_slow)
   END_RUNG
   RUNG wire#w1
      Move(in := 1, out1 => "PCS_2".MBmodeW_slow)
   END_RUNG
   RUNG wire#w1
      Move(in := 40861, out1 => "PCS_2".MBdataAddrW_slow)
   END_RUNG
   RUNG wire#w1
      Move(in := 2, out1 => "PCS_2".MBdataLenW_slow)
   END_RUNG
   // the same network as SCL:
   #_w1 := ("PCS_2".iCountDoneW_slow = 2) AND NOT "PCS_2".xREQW_slow;
   IF #_w1 THEN
       "PE_W_Block_GEN"(iType := 2, In_Data := "PCS_2".W, Out_Data => "PCS_2".arrDataW_slow);
       "PCS_2".MBmodeW_slow := 1;
       "PCS_2".MBdataAddrW_slow := 40861;
       "PCS_2".MBdataLenW_slow := 2;
   END_IF;
END_REGION

REGION Network 11: Write Bank DC Enable - to check
   RUNG wire#powerrail
      { S7_Templates := "SrcType := Int" } EQ_Contact(in1 := "PCS_2".iCountDoneW_slow, in2 := 3)
      Contact( "Reminder".x1 )
      I_Contact( "PCS_2".xREQW_slow )
      wire#w1
      Move(in := "PCS_2".W.wBankDcEnbCmd, out1 => "PCS_2".arrDataW_slow[1])
   END_RUNG
   RUNG wire#w1
      Move(in := 1, out1 => "PCS_2".MBmodeW_slow)
   END_RUNG
   RUNG wire#w1
      Move(in := 47052, out1 => "PCS_2".MBdataAddrW_slow)
   END_RUNG
   RUNG wire#w1
      Move(in := 1, out1 => "PCS_2".MBdataLenW_slow)
   END_RUNG
   // the same network as SCL:
   IF ("PCS_2".iCountDoneW_slow = 3) AND "Reminder".x1 AND NOT "PCS_2".xREQW_slow THEN
       "PCS_2".arrDataW_slow[1] := "PCS_2".W.wBankDcEnbCmd;
       "PCS_2".MBmodeW_slow := 1;
       "PCS_2".MBdataAddrW_slow := 47052;
       "PCS_2".MBdataLenW_slow := 1;
   END_IF;
END_REGION

REGION Network 12: Write Qac Reference
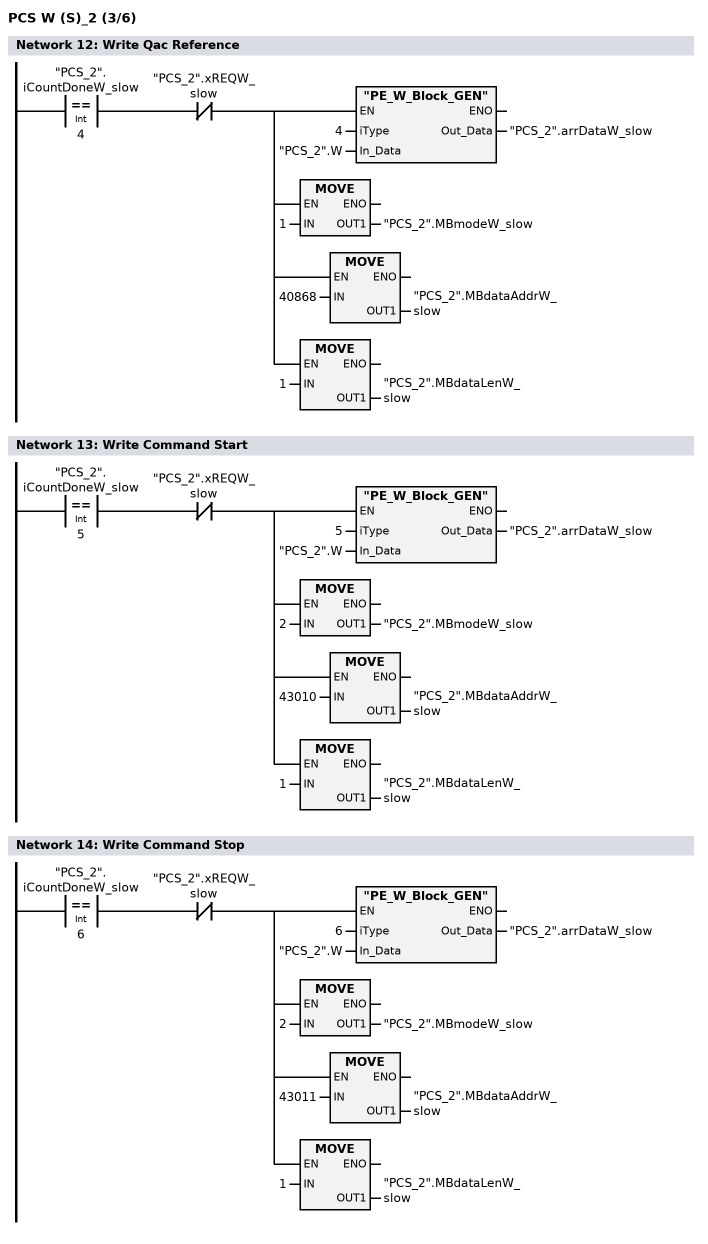
   RUNG wire#powerrail
      { S7_Templates := "SrcType := Int" } EQ_Contact(in1 := "PCS_2".iCountDoneW_slow, in2 := 4)
      I_Contact( "PCS_2".xREQW_slow )
      wire#w1
      "PE_W_Block_GEN"(iType := 4, In_Data := "PCS_2".W, Out_Data => "PCS_2".arrDataW_slow)
   END_RUNG
   RUNG wire#w1
      Move(in := 1, out1 => "PCS_2".MBmodeW_slow)
   END_RUNG
   RUNG wire#w1
      Move(in := 40868, out1 => "PCS_2".MBdataAddrW_slow)
   END_RUNG
   RUNG wire#w1
      Move(in := 1, out1 => "PCS_2".MBdataLenW_slow)
   END_RUNG
   // the same network as SCL:
   #_w1 := ("PCS_2".iCountDoneW_slow = 4) AND NOT "PCS_2".xREQW_slow;
   IF #_w1 THEN
       "PE_W_Block_GEN"(iType := 4, In_Data := "PCS_2".W, Out_Data => "PCS_2".arrDataW_slow);
       "PCS_2".MBmodeW_slow := 1;
       "PCS_2".MBdataAddrW_slow := 40868;
       "PCS_2".MBdataLenW_slow := 1;
   END_IF;
END_REGION

REGION Network 13: Write Command Start
   RUNG wire#powerrail
      { S7_Templates := "SrcType := Int" } EQ_Contact(in1 := "PCS_2".iCountDoneW_slow, in2 := 5)
      I_Contact( "PCS_2".xREQW_slow )
      wire#w1
      "PE_W_Block_GEN"(iType := 5, In_Data := "PCS_2".W, Out_Data => "PCS_2".arrDataW_slow)
   END_RUNG
   RUNG wire#w1
      Move(in := 2, out1 => "PCS_2".MBmodeW_slow)
   END_RUNG
   RUNG wire#w1
      Move(in := 43010, out1 => "PCS_2".MBdataAddrW_slow)
   END_RUNG
   RUNG wire#w1
      Move(in := 1, out1 => "PCS_2".MBdataLenW_slow)
   END_RUNG
   // the same network as SCL:
   #_w1 := ("PCS_2".iCountDoneW_slow = 5) AND NOT "PCS_2".xREQW_slow;
   IF #_w1 THEN
       "PE_W_Block_GEN"(iType := 5, In_Data := "PCS_2".W, Out_Data => "PCS_2".arrDataW_slow);
       "PCS_2".MBmodeW_slow := 2;
       "PCS_2".MBdataAddrW_slow := 43010;
       "PCS_2".MBdataLenW_slow := 1;
   END_IF;
END_REGION

REGION Network 14: Write Command Stop
   RUNG wire#powerrail
      { S7_Templates := "SrcType := Int" } EQ_Contact(in1 := "PCS_2".iCountDoneW_slow, in2 := 6)
      I_Contact( "PCS_2".xREQW_slow )
      wire#w1
      "PE_W_Block_GEN"(iType := 6, In_Data := "PCS_2".W, Out_Data => "PCS_2".arrDataW_slow)
   END_RUNG
   RUNG wire#w1
      Move(in := 2, out1 => "PCS_2".MBmodeW_slow)
   END_RUNG
   RUNG wire#w1
      Move(in := 43011, out1 => "PCS_2".MBdataAddrW_slow)
   END_RUNG
   RUNG wire#w1
      Move(in := 1, out1 => "PCS_2".MBdataLenW_slow)
   END_RUNG
   // the same network as SCL:
   #_w1 := ("PCS_2".iCountDoneW_slow = 6) AND NOT "PCS_2".xREQW_slow;
   IF #_w1 THEN
       "PE_W_Block_GEN"(iType := 6, In_Data := "PCS_2".W, Out_Data => "PCS_2".arrDataW_slow);
       "PCS_2".MBmodeW_slow := 2;
       "PCS_2".MBdataAddrW_slow := 43011;
       "PCS_2".MBdataLenW_slow := 1;
   END_IF;
END_REGION

REGION Network 15: Write Command Reset Fault
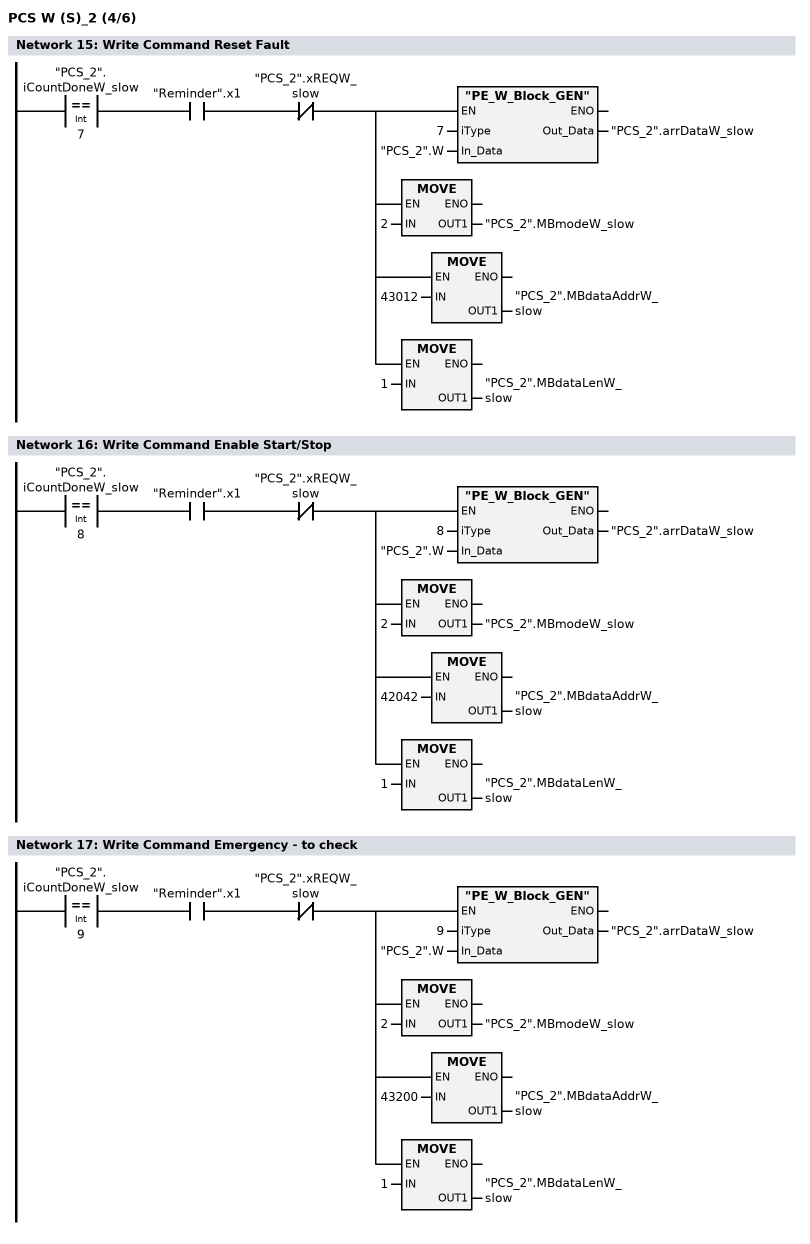
   RUNG wire#powerrail
      { S7_Templates := "SrcType := Int" } EQ_Contact(in1 := "PCS_2".iCountDoneW_slow, in2 := 7)
      Contact( "Reminder".x1 )
      I_Contact( "PCS_2".xREQW_slow )
      wire#w1
      "PE_W_Block_GEN"(iType := 7, In_Data := "PCS_2".W, Out_Data => "PCS_2".arrDataW_slow)
   END_RUNG
   RUNG wire#w1
      Move(in := 2, out1 => "PCS_2".MBmodeW_slow)
   END_RUNG
   RUNG wire#w1
      Move(in := 43012, out1 => "PCS_2".MBdataAddrW_slow)
   END_RUNG
   RUNG wire#w1
      Move(in := 1, out1 => "PCS_2".MBdataLenW_slow)
   END_RUNG
   // the same network as SCL:
   #_w1 := ("PCS_2".iCountDoneW_slow = 7) AND "Reminder".x1 AND NOT "PCS_2".xREQW_slow;
   IF #_w1 THEN
       "PE_W_Block_GEN"(iType := 7, In_Data := "PCS_2".W, Out_Data => "PCS_2".arrDataW_slow);
       "PCS_2".MBmodeW_slow := 2;
       "PCS_2".MBdataAddrW_slow := 43012;
       "PCS_2".MBdataLenW_slow := 1;
   END_IF;
END_REGION

REGION Network 16: Write Command Enable Start/Stop
   RUNG wire#powerrail
      { S7_Templates := "SrcType := Int" } EQ_Contact(in1 := "PCS_2".iCountDoneW_slow, in2 := 8)
      Contact( "Reminder".x1 )
      I_Contact( "PCS_2".xREQW_slow )
      wire#w1
      "PE_W_Block_GEN"(iType := 8, In_Data := "PCS_2".W, Out_Data => "PCS_2".arrDataW_slow)
   END_RUNG
   RUNG wire#w1
      Move(in := 2, out1 => "PCS_2".MBmodeW_slow)
   END_RUNG
   RUNG wire#w1
      Move(in := 42042, out1 => "PCS_2".MBdataAddrW_slow)
   END_RUNG
   RUNG wire#w1
      Move(in := 1, out1 => "PCS_2".MBdataLenW_slow)
   END_RUNG
   // the same network as SCL:
   #_w1 := ("PCS_2".iCountDoneW_slow = 8) AND "Reminder".x1 AND NOT "PCS_2".xREQW_slow;
   IF #_w1 THEN
       "PE_W_Block_GEN"(iType := 8, In_Data := "PCS_2".W, Out_Data => "PCS_2".arrDataW_slow);
       "PCS_2".MBmodeW_slow := 2;
       "PCS_2".MBdataAddrW_slow := 42042;
       "PCS_2".MBdataLenW_slow := 1;
   END_IF;
END_REGION

REGION Network 17: Write Command Emergency - to check
   RUNG wire#powerrail
      { S7_Templates := "SrcType := Int" } EQ_Contact(in1 := "PCS_2".iCountDoneW_slow, in2 := 9)
      Contact( "Reminder".x1 )
      I_Contact( "PCS_2".xREQW_slow )
      wire#w1
      "PE_W_Block_GEN"(iType := 9, In_Data := "PCS_2".W, Out_Data => "PCS_2".arrDataW_slow)
   END_RUNG
   RUNG wire#w1
      Move(in := 2, out1 => "PCS_2".MBmodeW_slow)
   END_RUNG
   RUNG wire#w1
      Move(in := 43200, out1 => "PCS_2".MBdataAddrW_slow)
   END_RUNG
   RUNG wire#w1
      Move(in := 1, out1 => "PCS_2".MBdataLenW_slow)
   END_RUNG
   // the same network as SCL:
   #_w1 := ("PCS_2".iCountDoneW_slow = 9) AND "Reminder".x1 AND NOT "PCS_2".xREQW_slow;
   IF #_w1 THEN
       "PE_W_Block_GEN"(iType := 9, In_Data := "PCS_2".W, Out_Data => "PCS_2".arrDataW_slow);
       "PCS_2".MBmodeW_slow := 2;
       "PCS_2".MBdataAddrW_slow := 43200;
       "PCS_2".MBdataLenW_slow := 1;
   END_IF;
END_REGION

REGION Network 18: Write WatchDog - to check
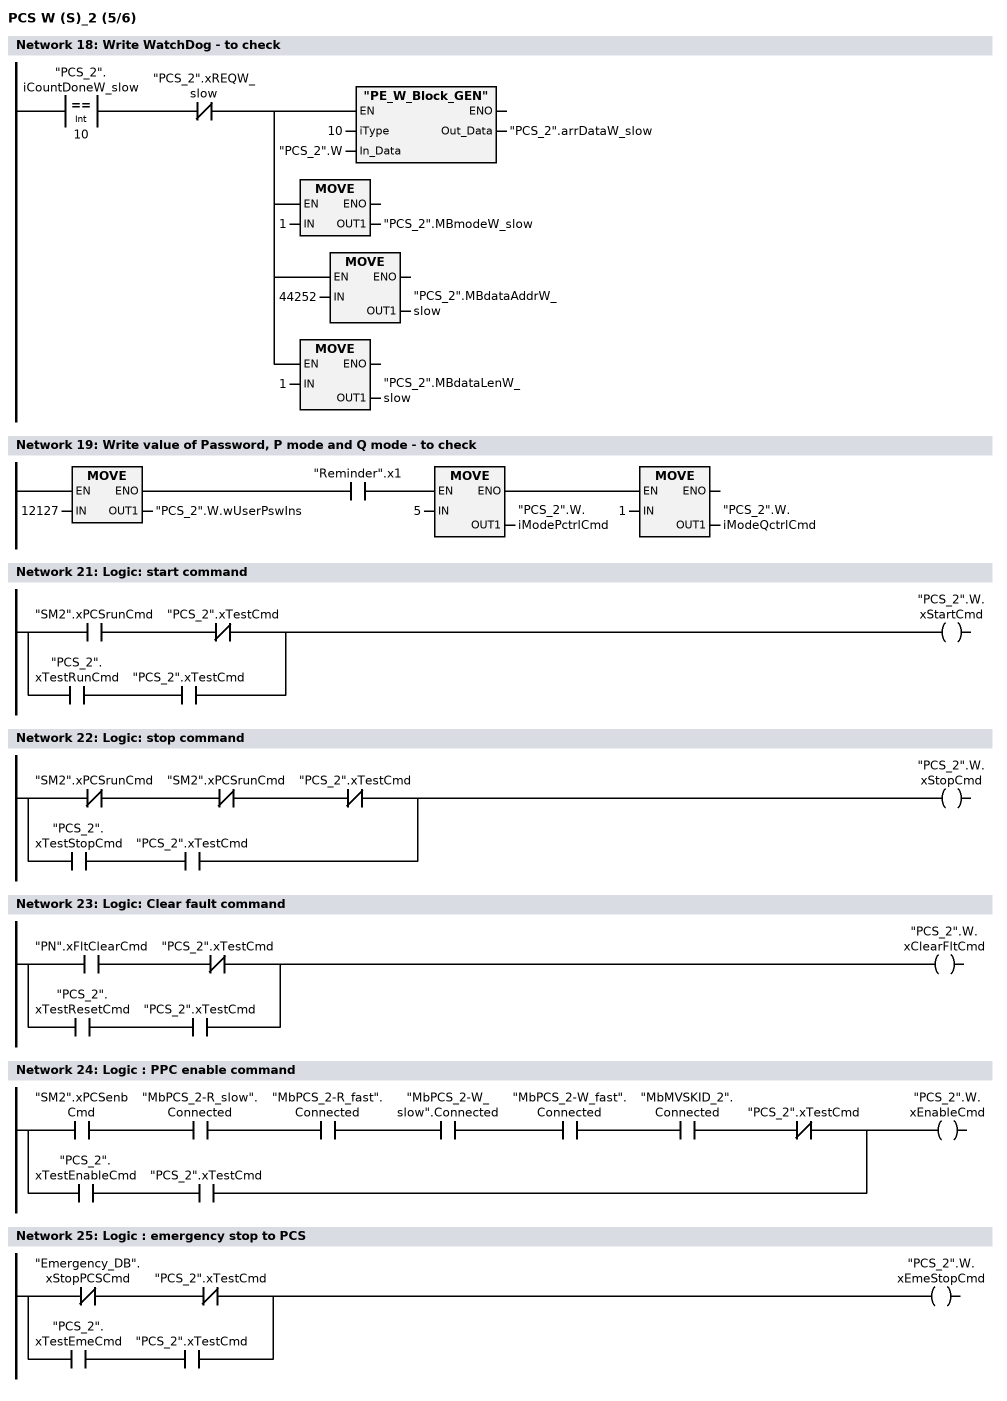
   RUNG wire#powerrail
      { S7_Templates := "SrcType := Int" } EQ_Contact(in1 := "PCS_2".iCountDoneW_slow, in2 := 10)
      I_Contact( "PCS_2".xREQW_slow )
      wire#w1
      "PE_W_Block_GEN"(iType := 10, In_Data := "PCS_2".W, Out_Data => "PCS_2".arrDataW_slow)
   END_RUNG
   RUNG wire#w1
      Move(in := 1, out1 => "PCS_2".MBmodeW_slow)
   END_RUNG
   RUNG wire#w1
      Move(in := 44252, out1 => "PCS_2".MBdataAddrW_slow)
   END_RUNG
   RUNG wire#w1
      Move(in := 1, out1 => "PCS_2".MBdataLenW_slow)
   END_RUNG
   // the same network as SCL:
   #_w1 := ("PCS_2".iCountDoneW_slow = 10) AND NOT "PCS_2".xREQW_slow;
   IF #_w1 THEN
       "PE_W_Block_GEN"(iType := 10, In_Data := "PCS_2".W, Out_Data => "PCS_2".arrDataW_slow);
       "PCS_2".MBmodeW_slow := 1;
       "PCS_2".MBdataAddrW_slow := 44252;
       "PCS_2".MBdataLenW_slow := 1;
   END_IF;
END_REGION

REGION Network 19: Write value of Password, P mode and Q mode - to check
   RUNG wire#powerrail
      Move(in := 12127, out1 => "PCS_2".W.wUserPswIns)
      Contact( "Reminder".x1 )
      Move(in := 5, out1 => "PCS_2".W.iModePctrlCmd)
      Move(in := 1, out1 => "PCS_2".W.iModeQctrlCmd)
   END_RUNG
   // the same network as SCL:
   "PCS_2".W.wUserPswIns := 12127;
   IF "Reminder".x1 THEN
       "PCS_2".W.iModePctrlCmd := 5;
       "PCS_2".W.iModeQctrlCmd := 1;
   END_IF;
END_REGION

REGION Network 21: Logic: start command
   RUNG wire#powerrail
      Contact( "SM2".xPCSrunCmd )
      I_Contact( "PCS_2".xTestCmd )
      wire#w1
      Coil( "PCS_2".W.xStartCmd )
   END_RUNG
   RUNG wire#powerrail
      Contact( "PCS_2".xTestRunCmd )
      Contact( "PCS_2".xTestCmd )
   END_RUNG wire#w1
   // the same network as SCL:
   "PCS_2".W.xStartCmd := ("SM2".xPCSrunCmd AND NOT "PCS_2".xTestCmd) OR ("PCS_2".xTestRunCmd AND "PCS_2".xTestCmd);
END_REGION

REGION Network 22: Logic: stop command
   RUNG wire#powerrail
      I_Contact( "SM2".xPCSrunCmd )
      I_Contact( "SM2".xPCSrunCmd )
      I_Contact( "PCS_2".xTestCmd )
      wire#w1
      Coil( "PCS_2".W.xStopCmd )
   END_RUNG
   RUNG wire#powerrail
      Contact( "PCS_2".xTestStopCmd )
      Contact( "PCS_2".xTestCmd )
   END_RUNG wire#w1
   // the same network as SCL:
   "PCS_2".W.xStopCmd := (NOT "SM2".xPCSrunCmd AND NOT "SM2".xPCSrunCmd AND NOT "PCS_2".xTestCmd) OR ("PCS_2".xTestStopCmd AND "PCS_2".xTestCmd);
END_REGION

REGION Network 23: Logic: Clear fault command
   RUNG wire#powerrail
      Contact( "PN".xFltClearCmd )
      I_Contact( "PCS_2".xTestCmd )
      wire#w1
      Coil( "PCS_2".W.xClearFltCmd )
   END_RUNG
   RUNG wire#powerrail
      Contact( "PCS_2".xTestResetCmd )
      Contact( "PCS_2".xTestCmd )
   END_RUNG wire#w1
   // the same network as SCL:
   "PCS_2".W.xClearFltCmd := ("PN".xFltClearCmd AND NOT "PCS_2".xTestCmd) OR ("PCS_2".xTestResetCmd AND "PCS_2".xTestCmd);
END_REGION

REGION Network 24: Logic : PPC enable command
   RUNG wire#powerrail
      Contact( "SM2".xPCSenbCmd )
      Contact( "MbPCS_2-R_slow".Connected )
      Contact( "MbPCS_2-R_fast".Connected )
      Contact( "MbPCS_2-W_slow".Connected )
      Contact( "MbPCS_2-W_fast".Connected )
      Contact( "MbMVSKID_2".Connected )
      I_Contact( "PCS_2".xTestCmd )
      wire#w1
      Coil( "PCS_2".W.xEnableCmd )
   END_RUNG
   RUNG wire#powerrail
      Contact( "PCS_2".xTestEnableCmd )
      Contact( "PCS_2".xTestCmd )
   END_RUNG wire#w1
   // the same network as SCL:
   "PCS_2".W.xEnableCmd := ("SM2".xPCSenbCmd AND "MbPCS_2-R_slow".Connected AND "MbPCS_2-R_fast".Connected AND "MbPCS_2-W_slow".Connected AND "MbPCS_2-W_fast".Connected AND "MbMVSKID_2".Connected AND NOT "PCS_2".xTestCmd) OR ("PCS_2".xTestEnableCmd AND "PCS_2".xTestCmd);
END_REGION

REGION Network 25: Logic : emergency stop to PCS
   RUNG wire#powerrail
      I_Contact( "Emergency_DB".xStopPCSCmd )
      I_Contact( "PCS_2".xTestCmd )
      wire#w1
      Coil( "PCS_2".W.xEmeStopCmd )
   END_RUNG
   RUNG wire#powerrail
      Contact( "PCS_2".xTestEmeCmd )
      Contact( "PCS_2".xTestCmd )
   END_RUNG wire#w1
   // the same network as SCL:
   "PCS_2".W.xEmeStopCmd := (NOT "Emergency_DB".xStopPCSCmd AND NOT "PCS_2".xTestCmd) OR ("PCS_2".xTestEmeCmd AND "PCS_2".xTestCmd);
END_REGION

REGION Network 26: G15.1.2 - Enable DCbus
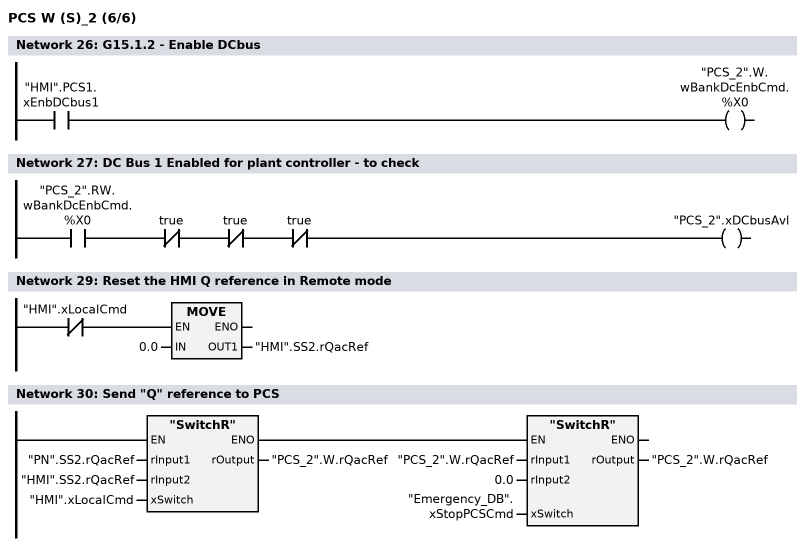
   RUNG wire#powerrail
      Contact( "HMI".PCS1.xEnbDCbus1 )
      Coil( "PCS_2".W.wBankDcEnbCmd.%X0 )
   END_RUNG
   // the same network as SCL:
   "PCS_2".W.wBankDcEnbCmd.%X0 := "HMI".PCS1.xEnbDCbus1;
END_REGION

REGION Network 27: DC Bus 1 Enabled for plant controller - to check
   RUNG wire#powerrail
      Contact( "PCS_2".RW.wBankDcEnbCmd.%X0 )
      I_Contact( true )
      I_Contact( true )
      I_Contact( true )
      Coil( "PCS_2".xDCbusAvl )
   END_RUNG
   // the same network as SCL:
   "PCS_2".xDCbusAvl := "PCS_2".RW.wBankDcEnbCmd.%X0 AND NOT true AND NOT true AND NOT true;
END_REGION

REGION Network 29: Reset the HMI Q reference in Remote mode
   RUNG wire#powerrail
      I_Contact( "HMI".xLocalCmd )
      Move(in := 0.0, out1 => "HMI".SS2.rQacRef)
   END_RUNG
   // the same network as SCL:
   IF NOT "HMI".xLocalCmd THEN "HMI".SS2.rQacRef := 0.0; END_IF;
END_REGION

REGION Network 30: Send "Q" reference to PCS
   RUNG wire#powerrail
      "SwitchR"(rInput1 := "PN".SS2.rQacRef, rInput2 := "HMI".SS2.rQacRef, xSwitch := "HMI".xLocalCmd, rOutput => "PCS_2".W.rQacRef)
      "SwitchR"(rInput1 := "PCS_2".W.rQacRef, rInput2 := 0.0, xSwitch := "Emergency_DB".xStopPCSCmd, rOutput => "PCS_2".W.rQacRef)
   END_RUNG
   // the same network as SCL:
   "SwitchR"(rInput1 := "PN".SS2.rQacRef,
             rInput2 := "HMI".SS2.rQacRef,
             xSwitch := "HMI".xLocalCmd,
             rOutput => "PCS_2".W.rQacRef,
             ENO => #_w1);
   IF #_w1 THEN
       "SwitchR"(rInput1 := "PCS_2".W.rQacRef,
                 rInput2 := 0.0,
                 xSwitch := "Emergency_DB".xStopPCSCmd,
                 rOutput => "PCS_2".W.rQacRef);
   END_IF;
END_REGION
END_FUNCTION

FUNCTION "test_1" : Void
{ S7_Optimized_Access := 'TRUE' }
VERSION : 0.1

BEGIN
END_FUNCTION

FUNCTION "SwitchI" : Void
{ S7_Optimized_Access := 'TRUE' }
VERSION : 0.1
   VAR_INPUT 
      rInput1 : Int;
      rInput2 : Int;
      xSwitch : Bool;
   END_VAR

   VAR_OUTPUT 
      rOutput : Int;
   END_VAR

   VAR_TEMP 
      rOutTemp : Int;
   END_VAR


BEGIN
	IF #xSwitch THEN
	    #rOutTemp := #rInput2;
	ELSE
	    #rOutTemp := #rInput1;
	END_IF;
	
	#rOutput := #rOutTemp;
END_FUNCTION

FUNCTION "SwitchS" : Void
{ S7_Optimized_Access := 'TRUE' }
VERSION : 0.1
   VAR_INPUT 
      rInput1 : String;
      rInput2 : String;
      xSwitch : Bool;
   END_VAR

   VAR_OUTPUT 
      rOutput : String;
   END_VAR

   VAR_TEMP 
      rOutTemp : String;
   END_VAR


BEGIN
	IF #xSwitch THEN
	    #rOutTemp := #rInput2;
	ELSE
	    #rOutTemp := #rInput1;
	END_IF;
	
	#rOutput := #rOutTemp;
END_FUNCTION

FUNCTION "SwitchW" : Void
{ S7_Optimized_Access := 'TRUE' }
VERSION : 0.1
   VAR_INPUT 
      rInput1 : Word;
      rInput2 : Word;
      xSwitch : Bool;
   END_VAR

   VAR_OUTPUT 
      rOutput : Word;
   END_VAR

   VAR_TEMP 
      rOutTemp : Word;
   END_VAR


BEGIN
	IF #xSwitch THEN
	    #rOutTemp := #rInput2;
	ELSE
	    #rOutTemp := #rInput1;
	END_IF;
	
	#rOutput := #rOutTemp;
END_FUNCTION

FUNCTION "Data" : Void
{ S7_Optimized_Access := 'TRUE' }
VERSION : 0.1
   VAR_TEMP 
      reminder : Bool;
   END_VAR


BEGIN
	
	// Data Battery Bank 1
	#reminder := "Reminder".x1; // da aggiungere rack 11-12
	"DashBoard".BB1.iNBRConn    := "BMS1".BB.iNBRconnectCount;
	"DashBoard".BB1.iTcellAvg   := "BMS1".BB.iTcellAvgMeas;
	"DashBoard".BB1.iTcellMax   := "BMS1".BB.iTcellMaxMeas;
	"DashBoard".BB1.iTcellMin   := "BMS1".BB.iTcellMinMeas;
	"DashBoard".BB1.rIdc        := "BMS1".BB.rIdcMeas;
	"DashBoard".BB1.rPdc        := ("BMS1".BB.rVdcMeas * "BMS1".BB.rIdcMeas);
	"DashBoard".BB1.rSOC        := "BMS1".BB.rSOCmeas;
	"DashBoard".BB1.rSOH        := "BMS1".BB.rSOHmeas;
	"DashBoard".BB1.rVcellAvg   := "BMS1".BB.rVcellAvgMeas;
	"DashBoard".BB1.rVcellMax   := "BMS1".BB.rVcellMaxMeas;
	"DashBoard".BB1.rVcellMin   := "BMS1".BB.rVcellMinMeas;
	"DashBoard".BB1.rVdc        := "BMS1".BB.rVdcMeas;
	
	// Data BB1 Rack 1
	
	"DashBoard".BB1BR1.iTamb        := "BMS1".BR01.iTambMeas;
	"DashBoard".BB1BR1.iTcellAvg    := "BMS1".BR01.iTcellAvgMeas;
	"DashBoard".BB1BR1.iTcellMax    := "BMS1".BR01.iTcellMaxMeas;
	"DashBoard".BB1BR1.iTmodMaxPos := "BMS1".BR01.iTmodMaxPos;
	"DashBoard".BB1BR1.iTcellMin    := "BMS1".BR01.iTcellMinMeas;
	"DashBoard".BB1BR1.iTmodMinPos := "BMS1".BR01.iTmodMinPos;
	"DashBoard".BB1BR1.iTempSet     := "BMS1".TMS01.iTempSet;
	"DashBoard".BB1BR1.iTrackIn     := "BMS1".BR01.iTrackInMeas;
	"DashBoard".BB1BR1.iTrackOut    := "BMS1".BR01.iTrackOutMeas;
	"DashBoard".BB1BR1.iVmodMaxPos := "BMS1".BR01.iVmodMaxPos;
	"DashBoard".BB1BR1.iVmodMinPos := "BMS1".BR01.iVmodMinPos;
	"DashBoard".BB1BR1.rIdc         := "BMS1".BR01.rIdcMeas;
	"DashBoard".BB1BR1.rSOC         := "BMS1".BR01.rSOCmeas;
	"DashBoard".BB1BR1.rSOH         := "BMS1".BR01.rSOHmeas;
	"DashBoard".BB1BR1.rVcellAvg    := "BMS1".BR01.rVcellAvgMeas;
	"DashBoard".BB1BR1.rVcellMax    := "BMS1".BR01.rVcellMaxMeas;
	"DashBoard".BB1BR1.rVcellMin    := "BMS1".BR01.rVcellMinMeas;
	"DashBoard".BB1BR1.rVdc         := "BMS1".BR01.rVdcMeas;
	
	// Data BB1 Rack 2
	
	"DashBoard".BB1BR2.iTamb        := "BMS1".BR02.iTambMeas;
	"DashBoard".BB1BR2.iTcellAvg    := "BMS1".BR02.iTcellAvgMeas;
	"DashBoard".BB1BR2.iTcellMax    := "BMS1".BR02.iTcellMaxMeas;
	"DashBoard".BB1BR2.iTmodMaxPos := "BMS1".BR02.iTmodMaxPos;
	"DashBoard".BB1BR2.iTcellMin    := "BMS1".BR02.iTcellMinMeas;
	"DashBoard".BB1BR2.iTmodMinPos := "BMS1".BR02.iTmodMinPos;
	"DashBoard".BB1BR2.iTempSet     := "BMS1".TMS02.iTempSet;
	"DashBoard".BB1BR2.iTrackIn     := "BMS1".BR02.iTrackInMeas;
	"DashBoard".BB1BR2.iTrackOut    := "BMS1".BR02.iTrackOutMeas;
	"DashBoard".BB1BR2.iVmodMaxPos := "BMS1".BR02.iVmodMaxPos;
	"DashBoard".BB1BR2.iVmodMinPos := "BMS1".BR02.iVmodMinPos;
	"DashBoard".BB1BR2.rIdc         := "BMS1".BR02.rIdcMeas;
	"DashBoard".BB1BR2.rSOC         := "BMS1".BR02.rSOCmeas;
	"DashBoard".BB1BR2.rSOH         := "BMS1".BR02.rSOHmeas;
	"DashBoard".BB1BR2.rVcellAvg    := "BMS1".BR02.rVcellAvgMeas;
	"DashBoard".BB1BR2.rVcellMax    := "BMS1".BR02.rVcellMaxMeas;
	"DashBoard".BB1BR2.rVcellMin    := "BMS1".BR02.rVcellMinMeas;
	"DashBoard".BB1BR2.rVdc         := "BMS1".BR02.rVdcMeas;
	
	// Data BB1 Rack 3
	
	"DashBoard".BB1BR3.iTamb        := "BMS1".BR03.iTambMeas;
	"DashBoard".BB1BR3.iTcellAvg    := "BMS1".BR03.iTcellAvgMeas;
	"DashBoard".BB1BR3.iTcellMax    := "BMS1".BR03.iTcellMaxMeas;
	"DashBoard".BB1BR3.iTmodMaxPos := "BMS1".BR03.iTmodMaxPos;
	"DashBoard".BB1BR3.iTcellMin    := "BMS1".BR03.iTcellMinMeas;
	"DashBoard".BB1BR3.iTmodMinPos := "BMS1".BR03.iTmodMinPos;
	"DashBoard".BB1BR3.iTempSet     := "BMS1".TMS03.iTempSet;
	"DashBoard".BB1BR3.iTrackIn     := "BMS1".BR03.iTrackInMeas;
	"DashBoard".BB1BR3.iTrackOut    := "BMS1".BR03.iTrackOutMeas;
	"DashBoard".BB1BR3.iVmodMaxPos := "BMS1".BR03.iVmodMaxPos;
	"DashBoard".BB1BR3.iVmodMinPos := "BMS1".BR03.iVmodMinPos;
	"DashBoard".BB1BR3.rIdc         := "BMS1".BR03.rIdcMeas;
	"DashBoard".BB1BR3.rSOC         := "BMS1".BR03.rSOCmeas;
	"DashBoard".BB1BR3.rSOH         := "BMS1".BR03.rSOHmeas;
	"DashBoard".BB1BR3.rVcellAvg    := "BMS1".BR03.rVcellAvgMeas;
	"DashBoard".BB1BR3.rVcellMax    := "BMS1".BR03.rVcellMaxMeas;
	"DashBoard".BB1BR3.rVcellMin    := "BMS1".BR03.rVcellMinMeas;
	"DashBoard".BB1BR3.rVdc         := "BMS1".BR03.rVdcMeas;
	
	// Data BB1 Rack 4
	
	"DashBoard".BB1BR4.iTamb        := "BMS1".BR04.iTambMeas;
	"DashBoard".BB1BR4.iTcellAvg    := "BMS1".BR04.iTcellAvgMeas;
	"DashBoard".BB1BR4.iTcellMax    := "BMS1".BR04.iTcellMaxMeas;
	"DashBoard".BB1BR4.iTmodMaxPos := "BMS1".BR04.iTmodMaxPos;
	"DashBoard".BB1BR4.iTcellMin    := "BMS1".BR04.iTcellMinMeas;
	"DashBoard".BB1BR4.iTmodMinPos := "BMS1".BR04.iTmodMinPos;
	"DashBoard".BB1BR4.iTempSet     := "BMS1".TMS04.iTempSet;
	"DashBoard".BB1BR4.iTrackIn     := "BMS1".BR04.iTrackInMeas;
	"DashBoard".BB1BR4.iTrackOut    := "BMS1".BR04.iTrackOutMeas;
	"DashBoard".BB1BR4.iVmodMaxPos := "BMS1".BR04.iVmodMaxPos;
	"DashBoard".BB1BR4.iVmodMinPos := "BMS1".BR04.iVmodMinPos;
	"DashBoard".BB1BR4.rIdc         := "BMS1".BR04.rIdcMeas;
	"DashBoard".BB1BR4.rSOC         := "BMS1".BR04.rSOCmeas;
	"DashBoard".BB1BR4.rSOH         := "BMS1".BR04.rSOHmeas;
	"DashBoard".BB1BR4.rVcellAvg    := "BMS1".BR04.rVcellAvgMeas;
	"DashBoard".BB1BR4.rVcellMax    := "BMS1".BR04.rVcellMaxMeas;
	"DashBoard".BB1BR4.rVcellMin    := "BMS1".BR04.rVcellMinMeas;
	"DashBoard".BB1BR4.rVdc         := "BMS1".BR04.rVdcMeas;
	
	// Data BB1 Rack 5
	
	"DashBoard".BB1BR5.iTamb        := "BMS1".BR05.iTambMeas;
	"DashBoard".BB1BR5.iTcellAvg    := "BMS1".BR05.iTcellAvgMeas;
	"DashBoard".BB1BR5.iTcellMax    := "BMS1".BR05.iTcellMaxMeas;
	"DashBoard".BB1BR5.iTmodMaxPos := "BMS1".BR05.iTmodMaxPos;
	"DashBoard".BB1BR5.iTcellMin    := "BMS1".BR05.iTcellMinMeas;
	"DashBoard".BB1BR5.iTmodMinPos := "BMS1".BR05.iTmodMinPos;
	"DashBoard".BB1BR5.iTempSet     := "BMS1".TMS05.iTempSet;
	"DashBoard".BB1BR5.iTrackIn     := "BMS1".BR05.iTrackInMeas;
	"DashBoard".BB1BR5.iTrackOut    := "BMS1".BR05.iTrackOutMeas;
	"DashBoard".BB1BR5.iVmodMaxPos := "BMS1".BR05.iVmodMaxPos;
	"DashBoard".BB1BR5.iVmodMinPos := "BMS1".BR05.iVmodMinPos;
	"DashBoard".BB1BR5.rIdc         := "BMS1".BR05.rIdcMeas;
	"DashBoard".BB1BR5.rSOC         := "BMS1".BR05.rSOCmeas;
	"DashBoard".BB1BR5.rSOH         := "BMS1".BR05.rSOHmeas;
	"DashBoard".BB1BR5.rVcellAvg    := "BMS1".BR05.rVcellAvgMeas;
	"DashBoard".BB1BR5.rVcellMax    := "BMS1".BR05.rVcellMaxMeas;
	"DashBoard".BB1BR5.rVcellMin    := "BMS1".BR05.rVcellMinMeas;
	"DashBoard".BB1BR5.rVdc         := "BMS1".BR05.rVdcMeas;
	
	// Data BB1 Rack 6
	
	"DashBoard".BB1BR6.iTamb        := "BMS1".BR06.iTambMeas;
	"DashBoard".BB1BR6.iTcellAvg    := "BMS1".BR06.iTcellAvgMeas;
	"DashBoard".BB1BR6.iTcellMax    := "BMS1".BR06.iTcellMaxMeas;
	"DashBoard".BB1BR6.iTmodMaxPos := "BMS1".BR06.iTmodMaxPos;
	"DashBoard".BB1BR6.iTcellMin    := "BMS1".BR06.iTcellMinMeas;
	"DashBoard".BB1BR6.iTmodMinPos := "BMS1".BR06.iTmodMinPos;
	"DashBoard".BB1BR6.iTempSet     := "BMS1".TMS06.iTempSet;
	"DashBoard".BB1BR6.iTrackIn     := "BMS1".BR06.iTrackInMeas;
	"DashBoard".BB1BR6.iTrackOut    := "BMS1".BR06.iTrackOutMeas;
	"DashBoard".BB1BR6.iVmodMaxPos := "BMS1".BR06.iVmodMaxPos;
	"DashBoard".BB1BR6.iVmodMinPos := "BMS1".BR06.iVmodMinPos;
	"DashBoard".BB1BR6.rIdc         := "BMS1".BR06.rIdcMeas;
	"DashBoard".BB1BR6.rSOC         := "BMS1".BR06.rSOCmeas;
	"DashBoard".BB1BR6.rSOH         := "BMS1".BR06.rSOHmeas;
	"DashBoard".BB1BR6.rVcellAvg    := "BMS1".BR06.rVcellAvgMeas;
	"DashBoard".BB1BR6.rVcellMax    := "BMS1".BR06.rVcellMaxMeas;
	"DashBoard".BB1BR6.rVcellMin    := "BMS1".BR06.rVcellMinMeas;
	"DashBoard".BB1BR6.rVdc         := "BMS1".BR06.rVdcMeas;
	
	// Data BB1 Rack 7
	
	"DashBoard".BB1BR7.iTamb        := "BMS1".BR07.iTambMeas;
	"DashBoard".BB1BR7.iTcellAvg    := "BMS1".BR07.iTcellAvgMeas;
	"DashBoard".BB1BR7.iTcellMax    := "BMS1".BR07.iTcellMaxMeas;
	"DashBoard".BB1BR7.iTmodMaxPos := "BMS1".BR07.iTmodMaxPos;
	"DashBoard".BB1BR7.iTcellMin    := "BMS1".BR07.iTcellMinMeas;
	"DashBoard".BB1BR7.iTmodMinPos := "BMS1".BR07.iTmodMinPos;
	"DashBoard".BB1BR7.iTempSet     := "BMS1".TMS07.iTempSet;
	"DashBoard".BB1BR7.iTrackIn     := "BMS1".BR07.iTrackInMeas;
	"DashBoard".BB1BR7.iTrackOut    := "BMS1".BR07.iTrackOutMeas;
	"DashBoard".BB1BR7.iVmodMaxPos := "BMS1".BR07.iVmodMaxPos;
	"DashBoard".BB1BR7.iVmodMinPos := "BMS1".BR07.iVmodMinPos;
	"DashBoard".BB1BR7.rIdc         := "BMS1".BR07.rIdcMeas;
	"DashBoard".BB1BR7.rSOC         := "BMS1".BR07.rSOCmeas;
	"DashBoard".BB1BR7.rSOH         := "BMS1".BR07.rSOHmeas;
	"DashBoard".BB1BR7.rVcellAvg    := "BMS1".BR07.rVcellAvgMeas;
	"DashBoard".BB1BR7.rVcellMax    := "BMS1".BR07.rVcellMaxMeas;
	"DashBoard".BB1BR7.rVcellMin    := "BMS1".BR07.rVcellMinMeas;
	"DashBoard".BB1BR7.rVdc         := "BMS1".BR07.rVdcMeas;
	
	// Data BB1 Rack 8
	
	"DashBoard".BB1BR8.iTamb        := "BMS1".BR08.iTambMeas;
	"DashBoard".BB1BR8.iTcellAvg    := "BMS1".BR08.iTcellAvgMeas;
	"DashBoard".BB1BR8.iTcellMax    := "BMS1".BR08.iTcellMaxMeas;
	"DashBoard".BB1BR8.iTmodMaxPos := "BMS1".BR08.iTmodMaxPos;
	"DashBoard".BB1BR8.iTcellMin    := "BMS1".BR08.iTcellMinMeas;
	"DashBoard".BB1BR8.iTmodMinPos := "BMS1".BR08.iTmodMinPos;
	"DashBoard".BB1BR8.iTempSet     := "BMS1".TMS08.iTempSet;
	"DashBoard".BB1BR8.iTrackIn     := "BMS1".BR08.iTrackInMeas;
	"DashBoard".BB1BR8.iTrackOut    := "BMS1".BR08.iTrackOutMeas;
	"DashBoard".BB1BR8.iVmodMaxPos := "BMS1".BR08.iVmodMaxPos;
	"DashBoard".BB1BR8.iVmodMinPos := "BMS1".BR08.iVmodMinPos;
	"DashBoard".BB1BR8.rIdc         := "BMS1".BR08.rIdcMeas;
	"DashBoard".BB1BR8.rSOC         := "BMS1".BR08.rSOCmeas;
	"DashBoard".BB1BR8.rSOH         := "BMS1".BR08.rSOHmeas;
	"DashBoard".BB1BR8.rVcellAvg    := "BMS1".BR08.rVcellAvgMeas;
	"DashBoard".BB1BR8.rVcellMax    := "BMS1".BR08.rVcellMaxMeas;
	"DashBoard".BB1BR8.rVcellMin    := "BMS1".BR08.rVcellMinMeas;
	"DashBoard".BB1BR8.rVdc         := "BMS1".BR08.rVdcMeas;
	
	// Data BB1 Rack 9
	
	"DashBoard".BB1BR9.iTamb        := "BMS1".BR09.iTambMeas;
	"DashBoard".BB1BR9.iTcellAvg    := "BMS1".BR09.iTcellAvgMeas;
	"DashBoard".BB1BR9.iTcellMax    := "BMS1".BR09.iTcellMaxMeas;
	"DashBoard".BB1BR9.iTmodMaxPos := "BMS1".BR09.iTmodMaxPos;
	"DashBoard".BB1BR9.iTcellMin    := "BMS1".BR09.iTcellMinMeas;
	"DashBoard".BB1BR9.iTmodMinPos := "BMS1".BR09.iTmodMinPos;
	"DashBoard".BB1BR9.iTempSet     := "BMS1".TMS09.iTempSet;
	"DashBoard".BB1BR9.iTrackIn     := "BMS1".BR09.iTrackInMeas;
	"DashBoard".BB1BR9.iTrackOut    := "BMS1".BR09.iTrackOutMeas;
	"DashBoard".BB1BR9.iVmodMaxPos := "BMS1".BR09.iVmodMaxPos;
	"DashBoard".BB1BR9.iVmodMinPos := "BMS1".BR09.iVmodMinPos;
	"DashBoard".BB1BR9.rIdc         := "BMS1".BR09.rIdcMeas;
	"DashBoard".BB1BR9.rSOC         := "BMS1".BR09.rSOCmeas;
	"DashBoard".BB1BR9.rSOH         := "BMS1".BR09.rSOHmeas;
	"DashBoard".BB1BR9.rVcellAvg    := "BMS1".BR09.rVcellAvgMeas;
	"DashBoard".BB1BR9.rVcellMax    := "BMS1".BR09.rVcellMaxMeas;
	"DashBoard".BB1BR9.rVcellMin    := "BMS1".BR09.rVcellMinMeas;
	"DashBoard".BB1BR9.rVdc         := "BMS1".BR09.rVdcMeas;
	
	// Data BB1 Rack 10
	
	"DashBoard".BB1BR10.iTamb           := "BMS1".BR10.iTambMeas;
	"DashBoard".BB1BR10.iTcellAvg       := "BMS1".BR10.iTcellAvgMeas;
	"DashBoard".BB1BR10.iTcellMax       := "BMS1".BR10.iTcellMaxMeas;
	"DashBoard".BB1BR10.iTmodMaxPos    := "BMS1".BR10.iTmodMaxPos;
	"DashBoard".BB1BR10.iTcellMin       := "BMS1".BR10.iTcellMinMeas;
	"DashBoard".BB1BR10.iTmodMinPos    := "BMS1".BR10.iTmodMinPos;
	"DashBoard".BB1BR10.iTempSet        := "BMS1".TMS10.iTempSet;
	"DashBoard".BB1BR10.iTrackIn        := "BMS1".BR10.iTrackInMeas;
	"DashBoard".BB1BR10.iTrackOut       := "BMS1".BR10.iTrackOutMeas;
	"DashBoard".BB1BR10.iVmodMaxPos    := "BMS1".BR10.iVmodMaxPos;
	"DashBoard".BB1BR10.iVmodMinPos    := "BMS1".BR10.iVmodMinPos;
	"DashBoard".BB1BR10.rIdc            := "BMS1".BR10.rIdcMeas;
	"DashBoard".BB1BR10.rSOC            := "BMS1".BR10.rSOCmeas;
	"DashBoard".BB1BR10.rSOH            := "BMS1".BR10.rSOHmeas;
	"DashBoard".BB1BR10.rVcellAvg       := "BMS1".BR10.rVcellAvgMeas;
	"DashBoard".BB1BR10.rVcellMax       := "BMS1".BR10.rVcellMaxMeas;
	"DashBoard".BB1BR10.rVcellMin       := "BMS1".BR10.rVcellMinMeas;
	"DashBoard".BB1BR10.rVdc            := "BMS1".BR10.rVdcMeas;
	
	// Data BB1 Rack 11
	
	"DashBoard".BB1BR11.iTamb := "BMS1".BR11.iTambMeas;
	"DashBoard".BB1BR11.iTcellAvg := "BMS1".BR11.iTcellAvgMeas;
	"DashBoard".BB1BR11.iTcellMax := "BMS1".BR11.iTcellMaxMeas;
	"DashBoard".BB1BR11.iTmodMaxPos := "BMS1".BR11.iTmodMaxPos;
	"DashBoard".BB1BR11.iTcellMin := "BMS1".BR11.iTcellMinMeas;
	"DashBoard".BB1BR11.iTmodMinPos := "BMS1".BR11.iTmodMinPos;
	"DashBoard".BB1BR11.iTempSet := "BMS1".TMS10.iTempSet;
	"DashBoard".BB1BR11.iTrackIn := "BMS1".BR11.iTrackInMeas;
	"DashBoard".BB1BR11.iTrackOut := "BMS1".BR11.iTrackOutMeas;
	"DashBoard".BB1BR11.iVmodMaxPos := "BMS1".BR11.iVmodMaxPos;
	"DashBoard".BB1BR11.iVmodMinPos := "BMS1".BR11.iVmodMinPos;
	"DashBoard".BB1BR11.rIdc := "BMS1".BR11.rIdcMeas;
	"DashBoard".BB1BR11.rSOC := "BMS1".BR11.rSOCmeas;
	"DashBoard".BB1BR11.rSOH := "BMS1".BR11.rSOHmeas;
	"DashBoard".BB1BR11.rVcellAvg := "BMS1".BR11.rVcellAvgMeas;
	"DashBoard".BB1BR11.rVcellMax := "BMS1".BR11.rVcellMaxMeas;
	"DashBoard".BB1BR11.rVcellMin := "BMS1".BR11.rVcellMinMeas;
	"DashBoard".BB1BR11.rVdc := "BMS1".BR11.rVdcMeas;
	
	// Data BB1 Rack 12
	
	"DashBoard".BB1BR12.iTamb := "BMS1".BR12.iTambMeas;
	"DashBoard".BB1BR12.iTcellAvg := "BMS1".BR12.iTcellAvgMeas;
	"DashBoard".BB1BR12.iTcellMax := "BMS1".BR12.iTcellMaxMeas;
	"DashBoard".BB1BR12.iTmodMaxPos := "BMS1".BR12.iTmodMaxPos;
	"DashBoard".BB1BR12.iTcellMin := "BMS1".BR12.iTcellMinMeas;
	"DashBoard".BB1BR12.iTmodMinPos := "BMS1".BR12.iTmodMinPos;
	"DashBoard".BB1BR12.iTempSet := "BMS1".TMS10.iTempSet;
	"DashBoard".BB1BR12.iTrackIn := "BMS1".BR12.iTrackInMeas;
	"DashBoard".BB1BR12.iTrackOut := "BMS1".BR12.iTrackOutMeas;
	"DashBoard".BB1BR12.iVmodMaxPos := "BMS1".BR12.iVmodMaxPos;
	"DashBoard".BB1BR12.iVmodMinPos := "BMS1".BR12.iVmodMinPos;
	"DashBoard".BB1BR12.rIdc := "BMS1".BR12.rIdcMeas;
	"DashBoard".BB1BR12.rSOC := "BMS1".BR12.rSOCmeas;
	"DashBoard".BB1BR12.rSOH := "BMS1".BR12.rSOHmeas;
	"DashBoard".BB1BR12.rVcellAvg := "BMS1".BR12.rVcellAvgMeas;
	"DashBoard".BB1BR12.rVcellMax := "BMS1".BR12.rVcellMaxMeas;
	"DashBoard".BB1BR12.rVcellMin := "BMS1".BR12.rVcellMinMeas;
	"DashBoard".BB1BR12.rVdc := "BMS1".BR12.rVdcMeas;
	
	// Data Battery Bank 2
	
	"DashBoard".BB2.iNBRConn    := "BMS2".BB.iNBRconnectCount;
	"DashBoard".BB2.iTcellAvg   := "BMS2".BB.iTcellAvgMeas;
	"DashBoard".BB2.iTcellMax   := "BMS2".BB.iTcellMaxMeas;
	"DashBoard".BB2.iTcellMin   := "BMS2".BB.iTcellMinMeas;
	"DashBoard".BB2.rIdc        := "BMS2".BB.rIdcMeas;
	"DashBoard".BB2.rPdc        := ("BMS2".BB.rVdcMeas * "BMS2".BB.rIdcMeas);
	"DashBoard".BB2.rSOC        := "BMS2".BB.rSOCmeas;
	"DashBoard".BB2.rSOH        := "BMS2".BB.rSOHmeas;
	"DashBoard".BB2.rVcellAvg   := "BMS2".BB.rVcellAvgMeas;
	"DashBoard".BB2.rVcellMax   := "BMS2".BB.rVcellMaxMeas;
	"DashBoard".BB2.rVcellMin   := "BMS2".BB.rVcellMinMeas;
	"DashBoard".BB2.rVdc        := "BMS2".BB.rVdcMeas;
	
	// Data BB2 Rack 1
	
	"DashBoard".BB2BR1.iTamb        := "BMS2".BR01.iTambMeas;
	"DashBoard".BB2BR1.iTcellAvg    := "BMS2".BR01.iTcellAvgMeas;
	"DashBoard".BB2BR1.iTcellMax    := "BMS2".BR01.iTcellMaxMeas;
	"DashBoard".BB2BR1.iTmodMaxPos := "BMS2".BR01.iTmodMaxPos;
	"DashBoard".BB2BR1.iTcellMin    := "BMS2".BR01.iTcellMinMeas;
	"DashBoard".BB2BR1.iTmodMinPos := "BMS2".BR01.iTmodMinPos;
	"DashBoard".BB2BR1.iTempSet     := "BMS2".TMS01.iTempSet;
	"DashBoard".BB2BR1.iTrackIn     := "BMS2".BR01.iTrackInMeas;
	"DashBoard".BB2BR1.iTrackOut    := "BMS2".BR01.iTrackOutMeas;
	"DashBoard".BB2BR1.iVmodMaxPos := "BMS2".BR01.iVmodMaxPos;
	"DashBoard".BB2BR1.iVmodMinPos := "BMS2".BR01.iVmodMinPos;
	"DashBoard".BB2BR1.rIdc         := "BMS2".BR01.rIdcMeas;
	"DashBoard".BB2BR1.rSOC         := "BMS2".BR01.rSOCmeas;
	"DashBoard".BB2BR1.rSOH         := "BMS2".BR01.rSOHmeas;
	"DashBoard".BB2BR1.rVcellAvg    := "BMS2".BR01.rVcellAvgMeas;
	"DashBoard".BB2BR1.rVcellMax    := "BMS2".BR01.rVcellMaxMeas;
	"DashBoard".BB2BR1.rVcellMin    := "BMS2".BR01.rVcellMinMeas;
	"DashBoard".BB2BR1.rVdc         := "BMS2".BR01.rVdcMeas;
	
	// Data BB2 Rack 2
	
	"DashBoard".BB2BR2.iTamb        := "BMS2".BR02.iTambMeas;
	"DashBoard".BB2BR2.iTcellAvg    := "BMS2".BR02.iTcellAvgMeas;
	"DashBoard".BB2BR2.iTcellMax    := "BMS2".BR02.iTcellMaxMeas;
	"DashBoard".BB2BR2.iTmodMaxPos := "BMS2".BR02.iTmodMaxPos;
	"DashBoard".BB2BR2.iTcellMin    := "BMS2".BR02.iTcellMinMeas;
	"DashBoard".BB2BR2.iTmodMinPos := "BMS2".BR02.iTmodMinPos;
	"DashBoard".BB2BR2.iTempSet     := "BMS2".TMS02.iTempSet;
	"DashBoard".BB2BR2.iTrackIn     := "BMS2".BR02.iTrackInMeas;
	"DashBoard".BB2BR2.iTrackOut    := "BMS2".BR02.iTrackOutMeas;
	"DashBoard".BB2BR2.iVmodMaxPos := "BMS2".BR02.iVmodMaxPos;
	"DashBoard".BB2BR2.iVmodMinPos := "BMS2".BR02.iVmodMinPos;
	"DashBoard".BB2BR2.rIdc         := "BMS2".BR02.rIdcMeas;
	"DashBoard".BB2BR2.rSOC         := "BMS2".BR02.rSOCmeas;
	"DashBoard".BB2BR2.rSOH         := "BMS2".BR02.rSOHmeas;
	"DashBoard".BB2BR2.rVcellAvg    := "BMS2".BR02.rVcellAvgMeas;
	"DashBoard".BB2BR2.rVcellMax    := "BMS2".BR02.rVcellMaxMeas;
	"DashBoard".BB2BR2.rVcellMin    := "BMS2".BR02.rVcellMinMeas;
	"DashBoard".BB2BR2.rVdc         := "BMS2".BR02.rVdcMeas;
	
	// Data BB2 Rack 3
	
	"DashBoard".BB2BR3.iTamb        := "BMS2".BR03.iTambMeas;
	"DashBoard".BB2BR3.iTcellAvg    := "BMS2".BR03.iTcellAvgMeas;
	"DashBoard".BB2BR3.iTcellMax    := "BMS2".BR03.iTcellMaxMeas;
	"DashBoard".BB2BR3.iTmodMaxPos := "BMS2".BR03.iTmodMaxPos;
	"DashBoard".BB2BR3.iTcellMin    := "BMS2".BR03.iTcellMinMeas;
	"DashBoard".BB2BR3.iTmodMinPos := "BMS2".BR03.iTmodMinPos;
	"DashBoard".BB2BR3.iTempSet     := "BMS2".TMS03.iTempSet;
	"DashBoard".BB2BR3.iTrackIn     := "BMS2".BR03.iTrackInMeas;
	"DashBoard".BB2BR3.iTrackOut    := "BMS2".BR03.iTrackOutMeas;
	"DashBoard".BB2BR3.iVmodMaxPos := "BMS2".BR03.iVmodMaxPos;
	"DashBoard".BB2BR3.iVmodMinPos := "BMS2".BR03.iVmodMinPos;
	"DashBoard".BB2BR3.rIdc         := "BMS2".BR03.rIdcMeas;
	"DashBoard".BB2BR3.rSOC         := "BMS2".BR03.rSOCmeas;
	"DashBoard".BB2BR3.rSOH         := "BMS2".BR03.rSOHmeas;
	"DashBoard".BB2BR3.rVcellAvg    := "BMS2".BR03.rVcellAvgMeas;
	"DashBoard".BB2BR3.rVcellMax    := "BMS2".BR03.rVcellMaxMeas;
	"DashBoard".BB2BR3.rVcellMin    := "BMS2".BR03.rVcellMinMeas;
	"DashBoard".BB2BR3.rVdc         := "BMS2".BR03.rVdcMeas;
	
	// Data BB2 Rack 4
	
	"DashBoard".BB2BR4.iTamb        := "BMS2".BR04.iTambMeas;
	"DashBoard".BB2BR4.iTcellAvg    := "BMS2".BR04.iTcellAvgMeas;
	"DashBoard".BB2BR4.iTcellMax    := "BMS2".BR04.iTcellMaxMeas;
	"DashBoard".BB2BR4.iTmodMaxPos := "BMS2".BR04.iTmodMaxPos;
	"DashBoard".BB2BR4.iTcellMin    := "BMS2".BR04.iTcellMinMeas;
	"DashBoard".BB2BR4.iTmodMinPos := "BMS2".BR04.iTmodMinPos;
	"DashBoard".BB2BR4.iTempSet     := "BMS2".TMS04.iTempSet;
	"DashBoard".BB2BR4.iTrackIn     := "BMS2".BR04.iTrackInMeas;
	"DashBoard".BB2BR4.iTrackOut    := "BMS2".BR04.iTrackOutMeas;
	"DashBoard".BB2BR4.iVmodMaxPos := "BMS2".BR04.iVmodMaxPos;
	"DashBoard".BB2BR4.iVmodMinPos := "BMS2".BR04.iVmodMinPos;
	"DashBoard".BB2BR4.rIdc         := "BMS2".BR04.rIdcMeas;
	"DashBoard".BB2BR4.rSOC         := "BMS2".BR04.rSOCmeas;
	"DashBoard".BB2BR4.rSOH         := "BMS2".BR04.rSOHmeas;
	"DashBoard".BB2BR4.rVcellAvg    := "BMS2".BR04.rVcellAvgMeas;
	"DashBoard".BB2BR4.rVcellMax    := "BMS2".BR04.rVcellMaxMeas;
	"DashBoard".BB2BR4.rVcellMin    := "BMS2".BR04.rVcellMinMeas;
	"DashBoard".BB2BR4.rVdc         := "BMS2".BR04.rVdcMeas;
	
	// Data BB2 Rack 5
	
	"DashBoard".BB2BR5.iTamb        := "BMS2".BR05.iTambMeas;
	"DashBoard".BB2BR5.iTcellAvg    := "BMS2".BR05.iTcellAvgMeas;
	"DashBoard".BB2BR5.iTcellMax    := "BMS2".BR05.iTcellMaxMeas;
	"DashBoard".BB2BR5.iTmodMaxPos := "BMS2".BR05.iTmodMaxPos;
	"DashBoard".BB2BR5.iTcellMin    := "BMS2".BR05.iTcellMinMeas;
	"DashBoard".BB2BR5.iTmodMinPos := "BMS2".BR05.iTmodMinPos;
	"DashBoard".BB2BR5.iTempSet     := "BMS2".TMS05.iTempSet;
	"DashBoard".BB2BR5.iTrackIn     := "BMS2".BR05.iTrackInMeas;
	"DashBoard".BB2BR5.iTrackOut    := "BMS2".BR05.iTrackOutMeas;
	"DashBoard".BB2BR5.iVmodMaxPos := "BMS2".BR05.iVmodMaxPos;
	"DashBoard".BB2BR5.iVmodMinPos := "BMS2".BR05.iVmodMinPos;
	"DashBoard".BB2BR5.rIdc         := "BMS2".BR05.rIdcMeas;
	"DashBoard".BB2BR5.rSOC         := "BMS2".BR05.rSOCmeas;
	"DashBoard".BB2BR5.rSOH         := "BMS2".BR05.rSOHmeas;
	"DashBoard".BB2BR5.rVcellAvg    := "BMS2".BR05.rVcellAvgMeas;
	"DashBoard".BB2BR5.rVcellMax    := "BMS2".BR05.rVcellMaxMeas;
	"DashBoard".BB2BR5.rVcellMin    := "BMS2".BR05.rVcellMinMeas;
	"DashBoard".BB2BR5.rVdc         := "BMS2".BR05.rVdcMeas;
	
	// Data BB2 Rack 6
	
	"DashBoard".BB2BR6.iTamb        := "BMS2".BR06.iTambMeas;
	"DashBoard".BB2BR6.iTcellAvg    := "BMS2".BR06.iTcellAvgMeas;
	"DashBoard".BB2BR6.iTcellMax    := "BMS2".BR06.iTcellMaxMeas;
	"DashBoard".BB2BR6.iTmodMaxPos := "BMS2".BR06.iTmodMaxPos;
	"DashBoard".BB2BR6.iTcellMin    := "BMS2".BR06.iTcellMinMeas;
	"DashBoard".BB2BR6.iTmodMinPos := "BMS2".BR06.iTmodMinPos;
	"DashBoard".BB2BR6.iTempSet     := "BMS2".TMS06.iTempSet;
	"DashBoard".BB2BR6.iTrackIn     := "BMS2".BR06.iTrackInMeas;
	"DashBoard".BB2BR6.iTrackOut    := "BMS2".BR06.iTrackOutMeas;
	"DashBoard".BB2BR6.iVmodMaxPos := "BMS2".BR06.iVmodMaxPos;
	"DashBoard".BB2BR6.iVmodMinPos := "BMS2".BR06.iVmodMinPos;
	"DashBoard".BB2BR6.rIdc         := "BMS2".BR06.rIdcMeas;
	"DashBoard".BB2BR6.rSOC         := "BMS2".BR06.rSOCmeas;
	"DashBoard".BB2BR6.rSOH         := "BMS2".BR06.rSOHmeas;
	"DashBoard".BB2BR6.rVcellAvg    := "BMS2".BR06.rVcellAvgMeas;
	"DashBoard".BB2BR6.rVcellMax    := "BMS2".BR06.rVcellMaxMeas;
	"DashBoard".BB2BR6.rVcellMin    := "BMS2".BR06.rVcellMinMeas;
	"DashBoard".BB2BR6.rVdc         := "BMS2".BR06.rVdcMeas;
	
	// Data BB2 Rack 7
	
	"DashBoard".BB2BR7.iTamb        := "BMS2".BR07.iTambMeas;
	"DashBoard".BB2BR7.iTcellAvg    := "BMS2".BR07.iTcellAvgMeas;
	"DashBoard".BB2BR7.iTcellMax    := "BMS2".BR07.iTcellMaxMeas;
	"DashBoard".BB2BR7.iTmodMaxPos := "BMS2".BR07.iTmodMaxPos;
	"DashBoard".BB2BR7.iTcellMin    := "BMS2".BR07.iTcellMinMeas;
	"DashBoard".BB2BR7.iTmodMinPos := "BMS2".BR07.iTmodMinPos;
	"DashBoard".BB2BR7.iTempSet     := "BMS2".TMS07.iTempSet;
	"DashBoard".BB2BR7.iTrackIn     := "BMS2".BR07.iTrackInMeas;
	"DashBoard".BB2BR7.iTrackOut    := "BMS2".BR07.iTrackOutMeas;
	"DashBoard".BB2BR7.iVmodMaxPos := "BMS2".BR07.iVmodMaxPos;
	"DashBoard".BB2BR7.iVmodMinPos := "BMS2".BR07.iVmodMinPos;
	"DashBoard".BB2BR7.rIdc         := "BMS2".BR07.rIdcMeas;
	"DashBoard".BB2BR7.rSOC         := "BMS2".BR07.rSOCmeas;
	"DashBoard".BB2BR7.rSOH         := "BMS2".BR07.rSOHmeas;
	"DashBoard".BB2BR7.rVcellAvg    := "BMS2".BR07.rVcellAvgMeas;
	"DashBoard".BB2BR7.rVcellMax    := "BMS2".BR07.rVcellMaxMeas;
	"DashBoard".BB2BR7.rVcellMin    := "BMS2".BR07.rVcellMinMeas;
	"DashBoard".BB2BR7.rVdc         := "BMS2".BR07.rVdcMeas;
	
	// Data BB2 Rack 8
	
	"DashBoard".BB2BR8.iTamb        := "BMS2".BR08.iTambMeas;
	"DashBoard".BB2BR8.iTcellAvg    := "BMS2".BR08.iTcellAvgMeas;
	"DashBoard".BB2BR8.iTcellMax    := "BMS2".BR08.iTcellMaxMeas;
	"DashBoard".BB2BR8.iTmodMaxPos := "BMS2".BR08.iTmodMaxPos;
	"DashBoard".BB2BR8.iTcellMin    := "BMS2".BR08.iTcellMinMeas;
	"DashBoard".BB2BR8.iTmodMinPos := "BMS2".BR08.iTmodMinPos;
	"DashBoard".BB2BR8.iTempSet     := "BMS2".TMS08.iTempSet;
	"DashBoard".BB2BR8.iTrackIn     := "BMS2".BR08.iTrackInMeas;
	"DashBoard".BB2BR8.iTrackOut    := "BMS2".BR08.iTrackOutMeas;
	"DashBoard".BB2BR8.iVmodMaxPos := "BMS2".BR08.iVmodMaxPos;
	"DashBoard".BB2BR8.iVmodMinPos := "BMS2".BR08.iVmodMinPos;
	"DashBoard".BB2BR8.rIdc         := "BMS2".BR08.rIdcMeas;
	"DashBoard".BB2BR8.rSOC         := "BMS2".BR08.rSOCmeas;
	"DashBoard".BB2BR8.rSOH         := "BMS2".BR08.rSOHmeas;
	"DashBoard".BB2BR8.rVcellAvg    := "BMS2".BR08.rVcellAvgMeas;
	"DashBoard".BB2BR8.rVcellMax    := "BMS2".BR08.rVcellMaxMeas;
	"DashBoard".BB2BR8.rVcellMin    := "BMS2".BR08.rVcellMinMeas;
	"DashBoard".BB2BR8.rVdc         := "BMS2".BR08.rVdcMeas;
	
	// Data BB2 Rack 9
	
	"DashBoard".BB2BR9.iTamb        := "BMS2".BR09.iTambMeas;
	"DashBoard".BB2BR9.iTcellAvg    := "BMS2".BR09.iTcellAvgMeas;
	"DashBoard".BB2BR9.iTcellMax    := "BMS2".BR09.iTcellMaxMeas;
	"DashBoard".BB2BR9.iTmodMaxPos := "BMS2".BR09.iTmodMaxPos;
	"DashBoard".BB2BR9.iTcellMin    := "BMS2".BR09.iTcellMinMeas;
	"DashBoard".BB2BR9.iTmodMinPos := "BMS2".BR09.iTmodMinPos;
	"DashBoard".BB2BR9.iTempSet     := "BMS2".TMS09.iTempSet;
	"DashBoard".BB2BR9.iTrackIn     := "BMS2".BR09.iTrackInMeas;
	"DashBoard".BB2BR9.iTrackOut    := "BMS2".BR09.iTrackOutMeas;
	"DashBoard".BB2BR9.iVmodMaxPos := "BMS2".BR09.iVmodMaxPos;
	"DashBoard".BB2BR9.iVmodMinPos := "BMS2".BR09.iVmodMinPos;
	"DashBoard".BB2BR9.rIdc         := "BMS2".BR09.rIdcMeas;
	"DashBoard".BB2BR9.rSOC         := "BMS2".BR09.rSOCmeas;
	"DashBoard".BB2BR9.rSOH         := "BMS2".BR09.rSOHmeas;
	"DashBoard".BB2BR9.rVcellAvg    := "BMS2".BR09.rVcellAvgMeas;
	"DashBoard".BB2BR9.rVcellMax    := "BMS2".BR09.rVcellMaxMeas;
	"DashBoard".BB2BR9.rVcellMin    := "BMS2".BR09.rVcellMinMeas;
	"DashBoard".BB2BR9.rVdc         := "BMS2".BR09.rVdcMeas;
	
	// Data BB2 Rack 10
	
	"DashBoard".BB2BR10.iTamb           := "BMS2".BR10.iTambMeas;
	"DashBoard".BB2BR10.iTcellAvg       := "BMS2".BR10.iTcellAvgMeas;
	"DashBoard".BB2BR10.iTcellMax       := "BMS2".BR10.iTcellMaxMeas;
	"DashBoard".BB2BR10.iTmodMaxPos    := "BMS2".BR10.iTmodMaxPos;
	"DashBoard".BB2BR10.iTcellMin       := "BMS2".BR10.iTcellMinMeas;
	"DashBoard".BB2BR10.iTmodMinPos    := "BMS2".BR10.iTmodMinPos;
	"DashBoard".BB2BR10.iTempSet        := "BMS2".TMS10.iTempSet;
	"DashBoard".BB2BR10.iTrackIn        := "BMS2".BR10.iTrackInMeas;
	"DashBoard".BB2BR10.iTrackOut       := "BMS2".BR10.iTrackOutMeas;
	"DashBoard".BB2BR10.iVmodMaxPos    := "BMS2".BR10.iVmodMaxPos;
	"DashBoard".BB2BR10.iVmodMinPos    := "BMS2".BR10.iVmodMinPos;
	"DashBoard".BB2BR10.rIdc            := "BMS2".BR10.rIdcMeas;
	"DashBoard".BB2BR10.rSOC            := "BMS2".BR10.rSOCmeas;
	"DashBoard".BB2BR10.rSOH            := "BMS2".BR10.rSOHmeas;
	"DashBoard".BB2BR10.rVcellAvg       := "BMS2".BR10.rVcellAvgMeas;
	"DashBoard".BB2BR10.rVcellMax       := "BMS2".BR10.rVcellMaxMeas;
	"DashBoard".BB2BR10.rVcellMin       := "BMS2".BR10.rVcellMinMeas;
	"DashBoard".BB2BR10.rVdc            := "BMS2".BR10.rVdcMeas;
	
	// Data BB2 Rack 11
	
	"DashBoard".BB2BR11.iTamb := "BMS2".BR11.iTambMeas;
	"DashBoard".BB2BR11.iTcellAvg := "BMS2".BR11.iTcellAvgMeas;
	"DashBoard".BB2BR11.iTcellMax := "BMS2".BR11.iTcellMaxMeas;
	"DashBoard".BB2BR11.iTmodMaxPos := "BMS2".BR11.iTmodMaxPos;
	"DashBoard".BB2BR11.iTcellMin := "BMS2".BR11.iTcellMinMeas;
	"DashBoard".BB2BR11.iTmodMinPos := "BMS2".BR11.iTmodMinPos;
	"DashBoard".BB2BR11.iTempSet := "BMS2".TMS10.iTempSet;
	"DashBoard".BB2BR11.iTrackIn := "BMS2".BR11.iTrackInMeas;
	"DashBoard".BB2BR11.iTrackOut := "BMS2".BR11.iTrackOutMeas;
	"DashBoard".BB2BR11.iVmodMaxPos := "BMS2".BR11.iVmodMaxPos;
	"DashBoard".BB2BR11.iVmodMinPos := "BMS2".BR11.iVmodMinPos;
	"DashBoard".BB2BR11.rIdc := "BMS2".BR11.rIdcMeas;
	"DashBoard".BB2BR11.rSOC := "BMS2".BR11.rSOCmeas;
	"DashBoard".BB2BR11.rSOH := "BMS2".BR11.rSOHmeas;
	"DashBoard".BB2BR11.rVcellAvg := "BMS2".BR11.rVcellAvgMeas;
	"DashBoard".BB2BR11.rVcellMax := "BMS2".BR11.rVcellMaxMeas;
	"DashBoard".BB2BR11.rVcellMin := "BMS2".BR11.rVcellMinMeas;
	"DashBoard".BB2BR11.rVdc := "BMS2".BR11.rVdcMeas;
	
	// Data BB2 Rack 12
	
	"DashBoard".BB2BR12.iTamb := "BMS2".BR12.iTambMeas;
	"DashBoard".BB2BR12.iTcellAvg := "BMS2".BR12.iTcellAvgMeas;
	"DashBoard".BB2BR12.iTcellMax := "BMS2".BR12.iTcellMaxMeas;
	"DashBoard".BB2BR12.iTmodMaxPos := "BMS2".BR12.iTmodMaxPos;
	"DashBoard".BB2BR12.iTcellMin := "BMS2".BR12.iTcellMinMeas;
	"DashBoard".BB2BR12.iTmodMinPos := "BMS2".BR12.iTmodMinPos;
	"DashBoard".BB2BR12.iTempSet := "BMS2".TMS10.iTempSet;
	"DashBoard".BB2BR12.iTrackIn := "BMS2".BR12.iTrackInMeas;
	"DashBoard".BB2BR12.iTrackOut := "BMS2".BR12.iTrackOutMeas;
	"DashBoard".BB2BR12.iVmodMaxPos := "BMS2".BR12.iVmodMaxPos;
	"DashBoard".BB2BR12.iVmodMinPos := "BMS2".BR12.iVmodMinPos;
	"DashBoard".BB2BR12.rIdc := "BMS2".BR12.rIdcMeas;
	"DashBoard".BB2BR12.rSOC := "BMS2".BR12.rSOCmeas;
	"DashBoard".BB2BR12.rSOH := "BMS2".BR12.rSOHmeas;
	"DashBoard".BB2BR12.rVcellAvg := "BMS2".BR12.rVcellAvgMeas;
	"DashBoard".BB2BR12.rVcellMax := "BMS2".BR12.rVcellMaxMeas;
	"DashBoard".BB2BR12.rVcellMin := "BMS2".BR12.rVcellMinMeas;
	"DashBoard".BB2BR12.rVdc := "BMS2".BR12.rVdcMeas;
	
	// Data PCS
	
	"DashBoard".PCS.DriveSt     := 0;
	"DashBoard".PCS.FreqRef     := 0.0;
	"DashBoard".PCS.Mref        := 0.0;
	"DashBoard".PCS.Nref        := 0.0;
	"DashBoard".PCS.OperMode    := 0;
	"DashBoard".PCS.Vref        := 0.0;
	//"DashBoard".PCS.iCodeSt     := "PCS_1".R.iCodeSt;
	//"DashBoard".PCS.rFreq       := "PCS_1".R.rFrMeas;
	//"DashBoard".PCS.rIdcBus1    := "PCS_1".R.rIdcBus1Meas;
	//"DashBoard".PCS.rIdcBus2    := "PCS1".R.rIdcBus2Meas;
	//"DashBoard".PCS.rIr         := "PCS1".R.rIrMeas;
	//"DashBoard".PCS.rIs         := "PCS1".R.rIsMeas;
	//"DashBoard".PCS.rIt         := "PCS1".R.rItMeas;
	//"DashBoard".PCS.rPac        := "PCS1".R.rPacMeas;
	//"DashBoard".PCS.rPacBus1Ref := "PCS1".W.rPac1Ref;
	//"DashBoard".PCS.rPacBus2Ref := "PCS1".W.rPac2Ref;
	//"DashBoard".PCS.rPdcBus1    := ("PCS1".R.rIdcBus1Meas * "PCS1".R.rVdcBus1Meas);
	//"DashBoard".PCS.rPdcBus2    := ("PCS1".R.rIdcBus2Meas * "PCS1".R.rVdcBus2Meas);
	//"DashBoard".PCS.rQac        := "PCS1".R.rQacMeas;
	//"DashBoard".PCS.rQacBus1Ref := "PCS1".W.rQac1Ref;
	//"DashBoard".PCS.rQacBus2Ref := "PCS1".W.rQac2Ref;
	//"DashBoard".PCS.rSac        := "PCS1".R.rSacMeas;
	//"DashBoard".PCS.rVdcBus1    := "PCS1".R.rVdcBus1Meas;
	//"DashBoard".PCS.rVdcBus2    := "PCS1".R.rVdcBus2Meas;
	//"DashBoard".PCS.rVrs        := "PCS1".R.rVrsMeas;
	//"DashBoard".PCS.rVst        := "PCS1".R.rVstMeas;
	//"DashBoard".PCS.rVtr        := "PCS1".R.rVtrMeas;
	
	// Data MVSKID
	
	//"SwitchI"(rInput1:= 0,
	//rInput2:= 1,
	//xSwitch:= "MV SKID".R.xLine1DiscCloseSt,
	//rOutput=> "DashBoard".MVSKID.iLine1DiscSt);
	
	//"SwitchI"(rInput1 := 0,
	     //     rInput2 := 1,
	     //     xSwitch := "MV SKID".R.xLine1GndCloseSt,
	     //     rOutput => "DashBoard".MVSKID.iLine1GroundSt);
	
	//"SwitchI"(rInput1 := 0,
	// rInput2 := 1,
	//  xSwitch := "MV SKID".R.xLine2DiscCloseSt,
	//   rOutput => "DashBoard".MVSKID.iLine2DiscSt);
	
	//"SwitchI"(rInput1 := 0,
	//      rInput2 := 1,
	//      xSwitch := "MV SKID".R.xLine2GndCloseSt,
	//      rOutput => "DashBoard".MVSKID.iLine2GroundSt);
	
	//"SwitchI"(rInput1 := 0,
	//   rInput2 := 1,
	//     xSwitch := "MV SKID".R.xProt1DiscCloseSt,
	//      rOutput => "DashBoard".MVSKID.iProt1DiscSt);
	
	//"SwitchI"(rInput1 := 0,
	//        rInput2 := 1,
	//        xSwitch := "MV SKID".R.xProt1GndCloseSt,
	//        rOutput => "DashBoard".MVSKID.iProt1GroundSt);
	
	//"SwitchI"(rInput1 := 0,
	//     rInput2 := 1,
	//      xSwitch := "MV SKID".R.xProt1CircBrkCloseSt,
	//      rOutput => "DashBoard".MVSKID.iProt1CircBrkSt);
	
	"DashBoard".MVSKID.rTempTrafo := 0.0;
	
	// Data State Machine
	
	"DashBoard".SM.iSS1 := "SM1".iCountSS;
	"DashBoard".SM.iSS2 := "SM2".iCountSS;
	
END_FUNCTION

FUNCTION "Init BMS" : Void
{ S7_Optimized_Access := 'TRUE' }
VERSION : 0.1

BEGIN
	        //CATL Modbus
	        //To run beetwen 10-20ms -> same as BMS 1 and BMS 2
	        
	        //BMS1 Initialized 10ms
	        
	        "BMS1".TCON10.InterfaceId := 64;
	        "BMS1".TCON10.ID := 1;
	        "BMS1".TCON10.RemoteAddress.ADDR[1] := 10;
	        "BMS1".TCON10.RemoteAddress.ADDR[2] := 138;
	        "BMS1".TCON10.RemoteAddress.ADDR[3] := 1;
	        "BMS1".TCON10.RemoteAddress.ADDR[4] := 31;
	        
	        "BMS1".TCON10.ActiveEstablished := true;
	        "BMS1".TCON10.ConnectionType := 11;
	        "BMS1".TCON10.RemotePort := 502;
	        
	        //BMS1 Initialized 10ms
	        
	        "BMS1".TCON11.InterfaceId := 64;
	        "BMS1".TCON11.ID := 2;
	        "BMS1".TCON11.RemoteAddress.ADDR[1] := 10;
	        "BMS1".TCON11.RemoteAddress.ADDR[2] := 138;
	        "BMS1".TCON11.RemoteAddress.ADDR[3] := 1;
	        "BMS1".TCON11.RemoteAddress.ADDR[4] := 31;
	        
	        "BMS1".TCON11.ActiveEstablished := true;
	        "BMS1".TCON11.ConnectionType := 11;
	        "BMS1".TCON11.RemotePort := 502;
	        
	        //BMS1 Initialized
	        
	        "BMS1".TCON.InterfaceId := 64;
	        "BMS1".TCON.ID := 3;
	        "BMS1".TCON.RemoteAddress.ADDR[1] := 10;
	        "BMS1".TCON.RemoteAddress.ADDR[2] := 138;
	        "BMS1".TCON.RemoteAddress.ADDR[3] := 1;
	        "BMS1".TCON.RemoteAddress.ADDR[4] := 31;
	        
	        "BMS1".TCON.ActiveEstablished := true;
	        "BMS1".TCON.ConnectionType := 11;
	        "BMS1".TCON.RemotePort := 502;
	        
	        //BMS2 Initialized 10ms
	        
	        "BMS2".TCON10.InterfaceId := 64;
	        "BMS2".TCON10.ID := 4;
	        "BMS2".TCON10.RemoteAddress.ADDR[1] := 10;
	        "BMS2".TCON10.RemoteAddress.ADDR[2] := 138;
	        "BMS2".TCON10.RemoteAddress.ADDR[3] := 1;
	        "BMS2".TCON10.RemoteAddress.ADDR[4] := 32;
	        
	        "BMS2".TCON10.ActiveEstablished := true;
	        "BMS2".TCON10.ConnectionType := 11;
	        "BMS2".TCON10.RemotePort := 502;
	        
	        //BMS2 Initialized 10ms
	        
	        "BMS2".TCON11.InterfaceId := 64;
	        "BMS2".TCON11.ID := 5;
	        "BMS2".TCON11.RemoteAddress.ADDR[1] := 10;
	        "BMS2".TCON11.RemoteAddress.ADDR[2] := 138;
	        "BMS2".TCON11.RemoteAddress.ADDR[3] := 1;
	        "BMS2".TCON11.RemoteAddress.ADDR[4] := 32;
	        
	        "BMS2".TCON11.ActiveEstablished := true;
	        "BMS2".TCON11.ConnectionType := 11;
	        "BMS2".TCON11.RemotePort := 502;
	        
	        //BMS2 Initialized
	        
	        "BMS2".TCON.InterfaceId := 64;
	        "BMS2".TCON.ID := 6;
	        "BMS2".TCON.RemoteAddress.ADDR[1] := 10;
	        "BMS2".TCON.RemoteAddress.ADDR[2] := 138;
	        "BMS2".TCON.RemoteAddress.ADDR[3] := 1;
	        "BMS2".TCON.RemoteAddress.ADDR[4] := 32;
	        
	        "BMS2".TCON.ActiveEstablished := true;
	        "BMS2".TCON.ConnectionType := 11;
	        "BMS2".TCON.RemotePort := 502;
	        
END_FUNCTION

FUNCTION "Init PE" : Void
{ S7_Optimized_Access := 'TRUE' }
VERSION : 0.1

BEGIN
	        //PCS (PE) Modbus
	        
	        //Initialized for read a 120 register at 10 ms
	        
	        "PCS_1".TCONR_fast.InterfaceId := 64;
	        "PCS_1".TCONR_fast.ID := 11;
	        "PCS_1".TCONR_fast.RemoteAddress.ADDR[1] := 10;
	        "PCS_1".TCONR_fast.RemoteAddress.ADDR[2] := 138;
	        "PCS_1".TCONR_fast.RemoteAddress.ADDR[3] := 1;
	        "PCS_1".TCONR_fast.RemoteAddress.ADDR[4] := 51;
	        
	        "PCS_1".TCONR_fast.ActiveEstablished := true;
	        "PCS_1".TCONR_fast.ConnectionType := 11;
	        "PCS_1".TCONR_fast.RemotePort := 502;
	        
	        //Initialized for read a writeble variables
	        
	        "PCS_1".TCONR_slow.InterfaceId := 64;
	        "PCS_1".TCONR_slow.ID := 12;
	        "PCS_1".TCONR_slow.RemoteAddress.ADDR[1] := 10;
	        "PCS_1".TCONR_slow.RemoteAddress.ADDR[2] := 138;
	        "PCS_1".TCONR_slow.RemoteAddress.ADDR[3] := 1;
	        "PCS_1".TCONR_slow.RemoteAddress.ADDR[4] := 51;
	        
	        "PCS_1".TCONR_slow.ActiveEstablished := true;
	        "PCS_1".TCONR_slow.ConnectionType := 11;
	        "PCS_1".TCONR_slow.RemotePort := 502;
	        
	        //Initialized for write a command
	        
	        "PCS_1".TCONW_slow.InterfaceId := 64;
	        "PCS_1".TCONW_slow.ID := 13;
	        "PCS_1".TCONW_slow.RemoteAddress.ADDR[1] := 10;
	        "PCS_1".TCONW_slow.RemoteAddress.ADDR[2] := 138;
	        "PCS_1".TCONW_slow.RemoteAddress.ADDR[3] := 1;
	        "PCS_1".TCONW_slow.RemoteAddress.ADDR[4] := 51;
	        
	        "PCS_1".TCONW_slow.ActiveEstablished := true;
	        "PCS_1".TCONW_slow.ConnectionType := 11;
	        "PCS_1".TCONW_slow.RemotePort := 502;
	        
	        
	        //MV SKID (PE) Modbus
	        
	        "MvSkid_1".TCON.InterfaceId := 64;
	        "MvSkid_1".TCON.ID := 14;
	        "MvSkid_1".TCON.RemoteAddress.ADDR[1] := 10;
	        "MvSkid_1".TCON.RemoteAddress.ADDR[2] := 138;
	        "MvSkid_1".TCON.RemoteAddress.ADDR[3] := 1;
	        "MvSkid_1".TCON.RemoteAddress.ADDR[4] := 53;
	        
	        "MvSkid_1".TCON.ActiveEstablished := true;
	        "MvSkid_1".TCON.ConnectionType := 11;
	        "MvSkid_1".TCON.RemotePort := 502;
	        
END_FUNCTION

FUNCTION "PN Read Data" : Void
{ S7_Optimized_Access := 'TRUE' }
VERSION : 0.1

BEGIN
	//******************************************************************//
	//                                                                  //
	//                      Read Data from PLC CORE                     //
	//                                                                  //
	//******************************************************************//
	
	//Boolean
	
	"PN".xStopCmd := "PN".R."x1.1";
	"PN".xStandByCmd := "PN".R."x1.2";
	"PN".xRunCmd := "PN".R."x1.3";
	"PN".xFltClearCmd := "PN".R."x1.4";
	"PN".xFltCmd := "PN".R."x1.8";
	
	"PN".MVSKID.xCircBrkCloseCmd := "PN".R."x2.1";
	"PN".MVSKID.xCircBrkOpenCmd := "PN".R."x2.2";
	"PN".MVSKID.xACDC_CloseCmd := "PN".R."x2.3";
	
	//Integer
	
	"PN".iKeepAlive := "PN".R.i1;
	
	//Real
	
	"PN".SS1.rPacRef := "PN".R.r1;
	"PN".SS1.rQacRef := "PN".R.r2;
	"PN".SS2.rPacRef := "PN".R.r3;
	"PN".SS2.rQacRef := "PN".R.r4;
	
END_FUNCTION

FUNCTION "PN Write Data" : Void
{ S7_Optimized_Access := 'TRUE' }
VERSION : 0.1

BEGIN
	//******************************************************************//
	//                                                                  //
	//                      Write Data from PLC CORE                    //
	//                                                                  //
	//******************************************************************//
	
	//Boolean
	
	"PN".W."x1.1" := "SS".xFltSt;
	"PN".W."x1.2" := "SS".xAlmSt;
	"PN".W."x1.3" := "SS".XWarSt;
	"PN".W."x1.4" := "MbMVSKID_1".Connected;
	"PN".W."x1.5" := "MbMVSKID_2".Connected;
	"PN".W."x1.6" := False;
	"PN".W."x1.7" := False;
	"PN".W."x1.8" := FALSE; ////to check prima c'era NAC system fire alert
	
	"PN".W."x2.1" := "BMS1".xBankAvl;
	"PN".W."x2.2" := "BMS1".xEnbCha;
	"PN".W."x2.3" := "BMS1".xEnbDsch;
	"PN".W."x2.4" := "BMS1".BBxFltSt;
	"PN".W."x2.5" := "BMS1".BBxAlmSt;
	"PN".W."x2.6" := "BMS1".BBxWarnSt;
	"PN".W."x2.7" := False;
	"PN".W."x2.8" := False;
	
	"PN".W."x3.1" := "BMS2".xBankAvl;
	"PN".W."x3.2" := "BMS2".xEnbCha;
	"PN".W."x3.3" := "BMS2".xEnbDsch;
	"PN".W."x3.4" := "BMS2".BBxFltSt;
	"PN".W."x3.5" := "BMS2".BBxAlmSt;
	"PN".W."x3.6" := "BMS2".BBxWarnSt;
	"PN".W."x3.7" := False;
	"PN".W."x3.8" := False;
	
	"PN".W."x4.1" := "PCS_1".xDCbusAvl;
	"PN".W."x4.2" := FALSE;
	"PN".W."x4.3" := "PCS_1".xLVRT;
	"PN".W."x4.4" := "PCS_1".xOVRT;
	"PN".W."x4.5" := "PCS_1".xFltSt;
	"PN".W."x4.6" := "PCS_1".xWarnSt;
	"PN".W."x4.7" := False;
	"PN".W."x4.8" := False;
	
	"PN".W."x5.1" := "MvSkid_1".xFltSt;
	"PN".W."x5.2" := "MvSkid_1".xAlmSt;
	"PN".W."x5.3" := "MvSkid_1".xWarnSt;
	"PN".W."x5.4" := False;
	"PN".W."x5.5" := False;
	"PN".W."x5.6" := False;
	"PN".W."x5.7" := False;
	"PN".W."x5.8" := False;
	
	//Integer
	
	"PN".W.i1 := "PN".R.i1;
	"PN".W.i2 := 0;
	
	"PN".W.i3.%B0   := INT_TO_BYTE("SM1".iCountSS);
	"PN".W.i3.%B1   := INT_TO_BYTE("SM2".iCountSS);
	"PN".W.i4       := 0;
	
	"PN".W.i5   := "BMS1".BB.iTcellMaxMeas;
	"PN".W.i6   := "BMS1".BB.iTcellAvgMeas;
	"PN".W.i7   := "BMS1".BB.iTcellMinMeas;
	"PN".W.i8   := "BMS1".BB.iNBRconnectCount;
	"PN".W.i9   := "BMS1".BB.iNBRtotalCount;
	"PN".W.i10  := WORD_TO_INT("BMS1".wRackOn);
	"PN".W.i11  := WORD_TO_INT("BMS1".wRackFlt);
	"PN".W.i12  := WORD_TO_INT("BMS1".BB.wSMstatusSt);
	"PN".W.i13  := 0;
	"PN".W.i14  := 0;
	
	"PN".W.i15  := "BMS2".BB.iTcellMaxMeas;
	"PN".W.i16  := "BMS2".BB.iTcellAvgMeas;
	"PN".W.i17  := "BMS2".BB.iTcellMinMeas;
	"PN".W.i18  := "BMS2".BB.iNBRconnectCount;
	"PN".W.i19  := "BMS2".BB.iNBRtotalCount;
	"PN".W.i20  := WORD_TO_INT("BMS2".wRackOn);;
	"PN".W.i21  := WORD_TO_INT("BMS2".wRackFlt);
	"PN".W.i22  := WORD_TO_INT("BMS2".BB.wSMstatusSt);
	"PN".W.i23  := 0;
	"PN".W.i24  := 0;
	
	"PN".W.i25  := "PCS_1".R.bStatusDspRJ14;
	"PN".W.i26  := WORD_TO_INT("PCS_1".W.wBankDcEnbCmd);
	"PN".W.i27  := 0;
	"PN".W.i28  := 0;
	"PN".W.i29  := 0;
	
	"PN".W.i30 := WORD_TO_INT("MvSkid_1".wLine1DiscSt);
	"PN".W.i31 := WORD_TO_INT("MvSkid_1".wLine2DiscSt);
	"PN".W.i32 := WORD_TO_INT("MvSkid_1".wProt1DiscSt);
	"PN".W.i33 := WORD_TO_INT("MvSkid_1".wProt1CircBrkSt);
	"PN".W.i34 := 0;
	"PN".W.i35 := 0;
	
	//Real
	
	"PN".W.r1   := "PCS_1".R.diCurrentFault;
	"PN".W.r2   := "PCS_1".R.diCurrentFaultModule;
	"PN".W.r3   := 0.0;
	"PN".W.r4   := 0.0;
	
	"PN".W.r5   := "BMS1".BB.rSOCmeas;
	"PN".W.r6   := "BMS1".BB.rSOHmeas;
	"PN".W.r7   := "BMS1".BB.rVdcMeas;
	"PN".W.r8   := "BMS1".BB.rIdcMeas;
	"PN".W.r9   := "BMS1".rPchaLim;
	"PN".W.r10  := "BMS1".rPdschLim;
	"PN".W.r11  := "BMS1".BB.rVcellMaxMeas;
	"PN".W.r12  := "BMS1".BB.rVcellAvgMeas;
	"PN".W.r13  := "BMS1".BB.rVcellMinMeas;
	"PN".W.r14  := 0.0;
	
	"PN".W.r15  := "BMS2".BB.rSOCmeas;
	"PN".W.r16  := "BMS2".BB.rSOHmeas;
	"PN".W.r17  := "BMS2".BB.rVdcMeas;
	"PN".W.r18  := "BMS2".BB.rIdcMeas;
	"PN".W.r19  := "BMS2".rPchaLim;
	"PN".W.r20  := "BMS2".rPdschLim;
	"PN".W.r21  := "BMS2".BB.rVcellMaxMeas;
	"PN".W.r22  := "BMS2".BB.rVcellAvgMeas;
	"PN".W.r23  := "BMS2".BB.rVcellMinMeas;
	"PN".W.r24  := 0.0;
	
	"PN".W.r25  := "PCS_1".rLVacMeas;
	"PN".W.r26  := "PCS_1".rIacTotMeas;
	"PN".W.r27  := "PCS_1".rPacBus1Meas;
	"PN".W.r28  := "PCS_1".rPacBus2Meas;
	"PN".W.r29  := "PCS_1".rQacBus1Meas;
	"PN".W.r30  := "PCS_1".rQacBus2Meas;
	"PN".W.r31  := "PCS_1".R.rDCvoltageBus_3;
	"PN".W.r32  := "PCS_1".R.rDCvoltageBus_4;
	"PN".W.r33  := "PCS_1".R.rDCvoltageExt_4;
	"PN".W.r34  := "PCS_1".R.rDCvoltageExt_2;
	"PN".W.r35  := "PCS_1".R.rDCvoltageLast_1;
	"PN".W.r36  := "PCS_1".R.rDCvoltageExt_3;
	"PN".W.r37  := "PCS_1".rMod1MaxTemp;
	"PN".W.r38  := "PCS_1".rMod2MaxTemp;
	"PN".W.r39  := "PCS_1".rMod3MaxTemp;
	"PN".W.r40  := "PCS_1".rMod4MaxTemp;
	"PN".W.r41  := "PCS_1".rMod5MaxTemp;
	"PN".W.r42  := "PCS_1".rMod6MaxTemp;
	"PN".W.r43  := 0.0;
	"PN".W.r44  := 0.0;
	
	"PN".W.r45 := "MvSkid_1".R.rPT100Trafo1St;
	"PN".W.r46 := 0.0;
	"PN".W.r47 := 0.0;
	
END_FUNCTION

FUNCTION "SM1_S1_Boot" : Void
{ S7_Optimized_Access := 'TRUE' }
VERSION : 0.1
   VAR_TEMP 
      xBoot_Ok : Bool;
      iT1 : S5Time;
   END_VAR


BEGIN
	// **********************************************************
	// *                   MANAGEMENT ACTION                    *
	// **********************************************************
	
	REGION State Machine Status
	    
	    "SM1".xSsBootSt      := True;
	    "SM1".xSsWarmUpSt    := False;
	    "SM1".xSsReadySt     := False;
	    "SM1".xSsStandBySt   := False;
	    "SM1".xSsRunSt       := False;
	    "SM1".xSsTestSt      := False;
	    "SM1".xSsAutoMaintSt := False;
	    "SM1".xSsStopSt      := False;
	    "SM1".xSsFaultSt     := False;
	    
	    "SM1".iCountSS := 1;
	    
	END_REGION
	
	REGION Wait PLC Status From Off to On
	    
	// When the PLC switch to Run after 5sec "xBootSt = True" and the transition "T1 = True"
	    
	#iT1 := S_ODT(
	    T_NO := 1,
	    S := "SM1".xRunPlcSt,
	    TV := S5T#5s,
	    Q => "SM1".xBootSt);
	END_REGION
	
	// **********************************************************
	// *                 MANAGEMENT TRANSITION                  *
	// **********************************************************
	
	// Transition from Boot to WarmUp
	
	IF "SM1".xBootSt
	THEN
	    "SM1".xT11 := True;
	    "SM1".xBootSt := False;
	END_IF;
	
END_FUNCTION

FUNCTION "SM1_S2_WarmUp" : Void
{ S7_Optimized_Access := 'TRUE' }
VERSION : 0.1
   VAR_TEMP 
      xWarmUpSt : Bool;
   END_VAR


BEGIN
	// **********************************************************
	// *                   MANAGEMENT ACTION                    *
	// **********************************************************
	
	REGION State Machine Status
	    
	    "SM1".xSsBootSt := False;
	    "SM1".xSsWarmUpSt := True;
	    "SM1".xSsReadySt := False;
	    "SM1".xSsStandBySt := False;
	    "SM1".xSsRunSt := False;
	    "SM1".xSsTestSt := False;
	    "SM1".xSsAutoMaintSt := False;
	    "SM1".xSsStopSt := False;
	    "SM1".xSsFaultSt := False;
	    
	    "SM1".iCountSS := 2;
	    
	END_REGION
	
	REGION Activation
	    
	    "SM1".xCommCmd := True;    //Enable all communication on the Power Island
	    "SM1".xAuxCmd := True;    //Enable all auxiliary equipment on the Power Island
	    
	END_REGION
	
	REGION Activation Active
	    
	    IF "SM1".xAuxSt AND "SM1".xCommSt     //Check the feedback of communication and auxiliary on the Power Island
	    THEN
	        #xWarmUpSt := True;
	        
	    END_IF;
	    
	END_REGION
	
	
	// **********************************************************
	// *                 MANAGEMENT TRANSITION                  *
	// **********************************************************
	
	// Transition from WarmUp to Ready
	
	IF #xWarmUpSt
	THEN
	    "SM1".xT21 := True;
	    #xWarmUpSt := False;
	END_IF;
	
	// Transition from WarmUp to Fault
	
	IF "SM1".xFltSt
	THEN
	    "SM1".xT22 := True;
	END_IF;
	
	// Reset Transition
	
	"SM1".xT11 := False;
	"SM1".xT81 := False;
	"SM1".xT91 := False;
	"SM1".xT74 := False;
	"SM1".xT75 := False;
	"SM1".xT76 := False;
	
END_FUNCTION

FUNCTION "SM1_S3_Ready" : Void
{ S7_Optimized_Access := 'TRUE' }
VERSION : 0.1
   VAR_TEMP 
      xSSysReadySt : Bool;
   END_VAR


BEGIN
	// **********************************************************
	// *                   MANAGEMENT ACTION                    *
	// **********************************************************
	
	REGION State Machine Status
	    
	    "SM1".xSsBootSt      := False;
	    "SM1".xSsWarmUpSt    := False;
	    "SM1".xSsReadySt     := True;
	    "SM1".xSsStandBySt   := False;
	    "SM1".xSsRunSt       := False;
	    "SM1".xSsTestSt      := False;
	    "SM1".xSsAutoMaintSt := False;
	    "SM1".xSsStopSt      := False;
	    "SM1".xSsFaultSt     := False;
	        
	    "SM1".iCountSS := 3;
	    
	END_REGION
	
	REGION Ready Condition
	    
	    IF "SM1".xReadyCondSt AND "SM1".xEnbSSysSt      //With ready condition and Subsystem enabled from HMI the subsystem is ready
	    THEN
	        #xSSysReadySt := True;
	    END_IF;
	    
	END_REGION
	
	REGION Command Battery Close
	    
	    IF #xSSysReadySt AND ("SM1".xStandByCmd OR "SM1".xRunCmd)       //With subsystem ready and standby or run command send close command to the battery
	    THEN
	        "SM1".xBattCloseCmd := True;
	    END_IF;
	    
	END_REGION
	
	REGION Command Enable PCS
	    
	    IF "SM1".xBattCloseSt AND "SM1".xMVbreakerCloseSt       //When the battery are closed and MV circuit breaker close send enable command to the PCS
	    THEN
	        "SM1".xPCSenbCmd := True;
	    END_IF;
	END_REGION
	
	
	// **********************************************************
	// *                 MANAGEMENT TRANSITION                  *
	// **********************************************************
	
	// Transition from Ready to StandBy
	
	IF "SM1".xBattCloseSt AND "SM1".xPCSreadySt     //With battery closed and PCS in ready condition go on standby state
	THEN
	    "SM1".xT31 := True;
	    #xSSysReadySt := False;
	END_IF;
	
	// Transition from Ready to Stop
	
	IF "SM1".xStopCmd AND False     //From ready status never go in stop state
	THEN
	    "SM1".xT32 := True;
	END_IF;
	
	// Transition from Ready to Fault
	
	IF "SM1".xFltSt     //With subsystem in fault go to the fault status
	THEN
	    "SM1".xT33 := True;
	END_IF;
	
	// Transition from Ready to Test
	
	IF "SM1".xTestCmd       //With test command from HMI go to the test state
	THEN
	    "SM1".xT34 := True;
	END_IF;
	
	// Reset Transition
	
	"SM1".xT21   := False;
	"SM1".xT61   := False;
	
END_FUNCTION

FUNCTION "SM1_S4_StandBy" : Void
{ S7_Optimized_Access := 'TRUE' }
VERSION : 0.1

BEGIN
	// **********************************************************
	// *                   MANAGEMENT ACTION                    *
	// **********************************************************
	
	REGION State Machine Status
	    
	    "SM1".xSsBootSt      := False;
	    "SM1".xSsWarmUpSt    := False;
	    "SM1".xSsReadySt     := False;
	    "SM1".xSsStandBySt   := True;
	    "SM1".xSsRunSt       := False;
	    "SM1".xSsTestSt      := False;
	    "SM1".xSsAutoMaintSt := False;
	    "SM1".xSsStopSt      := False;
	    "SM1".xSsFaultSt     := False;
	    
	    "SM1".iCountSS := 4;
	    
	END_REGION
	
	REGION Run Command
	    
	    IF "SM1".xRunCmd        //With run command send run command to the PCS
	    THEN
	        "SM1".xPCSrunCmd := True;
	    END_IF;
	    
	END_REGION
	
	
	// **********************************************************
	// *                 MANAGEMENT TRANSITION                  *
	// **********************************************************
	
	// Transition from StandBy to Run
	
	IF "SM1".xPCSrunSt AND "SM1".xRunCmd        //With PCS in run and the command on go to run state
	THEN
	    "SM1".xT41 := True;
	END_IF;
	
	// Transition from StandBy to AutoMaint
	
	IF "SM1".xAutomaintCmd      //With automaintenance command go to automaintenance state
	THEN
	    "SM1".xT42 := True;
	END_IF;
	
	// Transition from StandBy to Stop
	
	IF "SM1".xStopCmd OR NOT "SM1".xEnbSSysSt       //With stop command or subsystem not enabled go to stop state
	THEN
	    "SM1".xT43 := True;
	END_IF;
	
	// Transition from StandBy to Fault
	
	IF "SM1".xFltSt     //With subsystem in fault go to the fault state
	THEN
	    "SM1".xT44 := True;
	END_IF;
	
	// Reset Transition
	
	"SM1".xT31   := False;
	"SM1".xT51   := False;
	"SM1".xT71   := False;
	
END_FUNCTION

FUNCTION "SM1_S5_Run" : Void
{ S7_Optimized_Access := 'TRUE' }
VERSION : 0.1

BEGIN
	// **********************************************************
	// *                   MANAGEMENT ACTION                    *
	// **********************************************************
	
	REGION State Machine Status
	    
	    "SM1".xSsBootSt      := False;
	    "SM1".xSsWarmUpSt    := False;
	    "SM1".xSsReadySt     := False;
	    "SM1".xSsStandBySt   := False;
	    "SM1".xSsRunSt       := True;
	    "SM1".xSsTestSt      := False;
	    "SM1".xSsAutoMaintSt := False;
	    "SM1".xSsStopSt      := False;
	    "SM1".xSsFaultSt     := False;
	    
	    "SM1".iCountSS := 5;
	    
	END_REGION
	
	REGION StandBy Command
	    
	    IF "SM1".xStandByCmd        //With standby command send stop command to the PCS
	    THEN
	        "SM1".xPCSrunCmd := False;
	    END_IF;
	    
	END_REGION
	
	
	// **********************************************************
	// *                 MANAGEMENT TRANSITION                  *
	// **********************************************************
	
	// Transition from Run to StandBy
	
	IF "SM1".xStandByCmd AND "SM1".xPCSreadySt      //With standby command e PCS in ready return to standby state
	THEN
	    "SM1".xT51 := True;
	END_IF;
	
	// Transition from Run to Stop
	
	IF "SM1".xStopCmd OR NOT "SM1".xEnbSSysSt       //With stop command or subsystem not enabled go to stop state
	THEN
	    "SM1".xT52 := True;
	END_IF;
	
	// Transition from Run to Fault
	
	IF "SM1".xFltSt     //With subsystem in fault go to the fault state
	THEN
	    "SM1".xT53 := True;
	END_IF;
	
	// Reset Transition
	
	"SM1".xT41 := False;
	
END_FUNCTION

FUNCTION "SM1_S6_Test" : Void
{ S7_Optimized_Access := 'TRUE' }
VERSION : 0.1

BEGIN
	// **********************************************************
	// *                   MANAGEMENT ACTION                    *
	// **********************************************************
	
	REGION State Machine Status
	    
	    "SM1".xSsBootSt := False;
	    "SM1".xSsWarmUpSt := False;
	    "SM1".xSsReadySt := False;
	    "SM1".xSsStandBySt := False;
	    "SM1".xSsRunSt := False;
	    "SM1".xSsTestSt := True;
	    "SM1".xSsAutoMaintSt := False;
	    "SM1".xSsStopSt := False;
	    "SM1".xSsFaultSt := False;
	    
	    "SM1".iCountSS := 6;
	    
	END_REGION
	
	"SM1".xPCSrunCmd := False;      //All command in this state are not necessary but only for safety
	
	REGION PCS enable Off
	    
	    IF "SM1".xPCSreadySt
	    THEN
	        "SM1".xPCSenbCmd := False;
	    END_IF;
	END_REGION
	
	REGION Command Open Battery
	    
	    IF "SM1".xPCSstopSt
	    THEN
	        "SM1".xBattCloseCmd := False;
	    END_IF;
	END_REGION
	
	
	// **********************************************************
	// *                 MANAGEMENT TRANSITION                  *
	// **********************************************************
	
	// Transition from Test to Ready
	
	IF NOT "SM1".xTestCmd       //Without test command return to ready state
	THEN
	    "SM1".xT61 := True;
	END_IF;
	
	// Transition from Test to Fault
	
	IF "SM1".xFltSt     //With subsystem in fault go to the fault state
	THEN
	    "SM1".xT62 := True;
	END_IF;
	
	// Reset Transition
	
	"SM1".xT34 := False;
	
END_FUNCTION

FUNCTION "SM1_S7_AutoMaint" : Void
{ S7_Optimized_Access := 'TRUE' }
VERSION : 0.1

BEGIN
	// **********************************************************
	// *                   MANAGEMENT ACTION                    *
	// **********************************************************
	
	REGION State Machine Status
	    
	    "SM1".xSsBootSt      := False;
	    "SM1".xSsWarmUpSt    := False;
	    "SM1".xSsReadySt     := False;
	    "SM1".xSsStandBySt   := False;
	    "SM1".xSsRunSt       := False;
	    "SM1".xSsTestSt      := False;
	    "SM1".xSsAutoMaintSt := True;
	    "SM1".xSsStopSt      := False;
	    "SM1".xSsFaultSt     := False;
	    
	    "SM1".iCountSS := 7;
	    
	END_REGION
	
	REGION Autocharge Bank
	    
	    "SM1".xPCSrunCmd := True;       //In automaintenance state send run command to the PCS
	    
	    IF "SM1".xPCSrunSt      //When PCS are in run read the active power reference from HMI
	    THEN
	        "SM1".rPacAutomRef := "HMI".rPacAutomRef;
	    END_IF;
	    
	END_REGION
	
	
	// **********************************************************
	// *                 MANAGEMENT TRANSITION                  *
	// **********************************************************
	
	// Transition from AutoMaint to StandBy
	
	IF "SM1".xAutomaintSt       //Without automaintenance command from battery return to standby state
	THEN
	    "SM1".xT71 := True;
	END_IF;
	
	// Transition from AutoMaint to Stop
	
	IF "SM1".xStopCmd       //With stop command go to stop state
	THEN
	    "SM1".xT72 := True;
	END_IF;
	
	// Transition from AutoMaint to Fault
	
	IF "SM1".xFltSt     //With subsystem in fault go to the fault state
	THEN
	    "SM1".xT73 := True;
	END_IF;
	
	// Reset Transition
	
	"SM1".xT42    := False;
	
END_FUNCTION

FUNCTION "SM1_S8_Stop" : Void
{ S7_Optimized_Access := 'TRUE' }
VERSION : 0.1

BEGIN
	// **********************************************************
	// *                   MANAGEMENT ACTION                    *
	// **********************************************************
	
	REGION State Machine Status
	    
	    "SM1".xSsBootSt      := False;
	    "SM1".xSsWarmUpSt    := False;
	    "SM1".xSsReadySt     := False;
	    "SM1".xSsStandBySt   := False;
	    "SM1".xSsRunSt       := False;
	    "SM1".xSsTestSt      := False;
	    "SM1".xSsAutoMaintSt := False;
	    "SM1".xSsStopSt      := True;
	    "SM1".xSsFaultSt     := False;
	    
	    "SM1".iCountSS := 8;
	    
	END_REGION
	
	"SM1".xPCSrunCmd := False;      //In stop state send stop command to the PCS
	
	REGION PCS enable Off
	    
	    IF "SM1".xPCSreadySt        //When the PCS are in ready take out the enable command to the PCS
	    THEN
	        "SM1".xPCSenbCmd := False;
	    END_IF;
	END_REGION
	
	REGION Command Open Battery
	    
	    IF "SM1".xPCSstopSt     //When the PCS are in stop send open command to the battery
	    THEN
	        "SM1".xBattCloseCmd := False;
	    END_IF;
	END_REGION
	
	
